ABB RobotStudio station: Topsy_Turvey_Pack_N_Go_RW_5.16.rspag

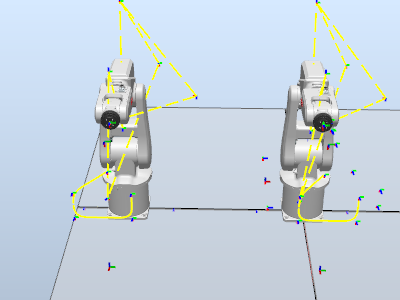
--- station ---
Station Turvey_Solution_2 (saved by RobotStudio 24.2.10789.0)
Controller 120-502354_Topsy, task T_ROB1: task frame (RAPID world) sits at (0, -769, 0) mm in the station
Controller 120-501650_Turvey
  mechanical unit ROB_1: IRB120_Turvey, 6 joints, base frame (0, 0, 0) mm
Controller 120-502354_Topsy
  mechanical unit ROB_1: IRB120_Topsy, 6 joints, base frame (0, 0, 0) mm
Layout (positions relative to the parent item):
  - IRB120_Turvey [mechanism, from %ABB.RobotStudio.Models.IRB120%\IRB120_3_58_G_01.rslib] at (0, 0, 0) mm; joint values [0, 0, 0, 0, 0, 0] (rad or m)
  - IRB120_Topsy [mechanism, from %ABB.RobotStudio.Models.IRB120%\IRB120_3_58_G_01.rslib] at (0, -769, 0) mm; joint values [0, 0, 0, 0, 0, 0] (rad or m)
Targets, tools, work objects and paths stored in the station and not in the controller backup, written as RAPID:
! task T_ROB1
MODULE MainModule
  CONST robtarget pos1:=[[366.18,1.37,632.09],[0.674845,-0.0204665,0.737511,-0.015567],[0,0,-1,0],[9E+09,9E+09,9E+09,9E+09,9E+09,9E+09]];
  CONST jointtarget JtCalpos:=[[0,0,0,0,0,0],[9E+09,9E+09,9E+09,9E+09,0,9E+09]];
  CONST jointtarget JtHome:=[[0,0,0,90,0,0],[9E+09,9E+09,9E+09,9E+09,0,9E+09]];
  PROC R_Home()
    WaitTime 5;
    WaitTime 5;
    MoveAbsJ jHomePos,v500,fine,tool0;
  ENDPROC
  PROC R_Storage()
    WaitTime 5;
    WaitTime 5;
    MoveAbsJ jStorage,v500,fine,tool0;
  ENDPROC
ENDMODULE

! task T_ROB1
MODULE MainModule
  PROC R_Home()
    WaitTime 5;
    WaitTime 5;
    MoveAbsJ jHomePos,v500,fine,tool0;
  ENDPROC
  PROC R_Storage()
    WaitTime 5;
    WaitTime 5;
    MoveAbsJ jStorage,v500,fine,tool0;
  ENDPROC
ENDMODULE


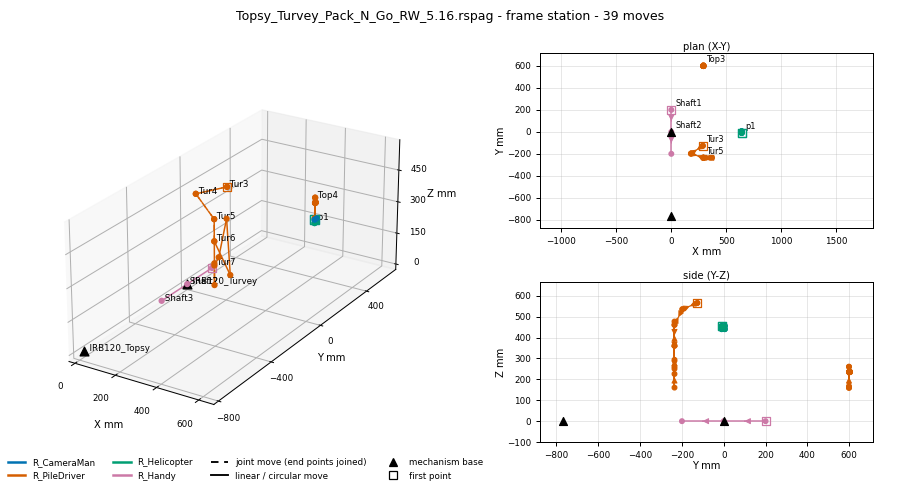
[picture p0: tool path of Topsy_Turvey_Pack_N_Go_RW_5.16.rspag in frame station, 39 of 203 moves have a stored position in this frame; points joined in program order, loops and branches not executed]
--- Backups/120-501650_Turvey/RAPID/TASK1/PROGMOD/MainModule.mod ---
MODULE MainModule
    !    !*****************************************************
    !    !Module Name:   MainModule
    !    !Version:       1.22
    !    !Description:   Main Module
    !    !Date:          2024-08-01
    !    !Author:        @ManicZanic
    !    !*****************************************************
    !    !Change Log:
    !    !2024-08-01:    @ManicZanic - Orignal core structure developed
    !    !2024-08-21:    @ManicZanic - Moved non TOH routines to Main module.
    !    !                           - Added Menu options to all routines.
    !    !                           - Added NCameraLoop to disconnect variables from other modules
    !    !                           - Cleaned up text a bit
    !    !                           - Formatted text
    !    !                           - Added Yoga Pose positions
    !    !                           - Added blank JustDance program
    !    !2024-08-22:    @ManicZanic - Removed unused code
    !    !                           - Removed task specific ToolData
    !    !2024-08-22:    @ManicZanic - Programmed DancingQueen routine.
    !    !                           - Programmed YogaPose routine
    !    !                           - Edited menu names
    !    !2024-08-26:    @ManicZanic - Modified motion alert notification interface.
    !    !                           - Created universal speed selection progam
    !    !                           - Modified Yoga Poses
    !    !2024-08-29:    @ManicZanic - Updated UI to add option for no motion alarm and to edit menus
    !    !*****************************************************

    PERS bool bMenu:=TRUE;
    PERS bool bTopsy:=FALSE;
    PERS bool bTurvey:=TRUE;
    PERS bool CondomMode:=FALSE;
    PERS bool RawDogMode:=TRUE;

    !CURRENT VELOCITY
    VAR speeddata VSpeed:=V300;

    VAR num ERR_TP_DOBREAK;
    !VAR num CurrentIndex:=nMenuOption;
    VAR num nMenuOption;

    VAR btnres answer;

    CONST string LoopMessage{5}:=[" "," ","Enter How Many Times To Loop Dance Program"," ","0=INFINITE"];
    CONST string CautionMessage{5}:=[" "," "," ","Press RUN to continue","Press CANCEL to return to previous menu"];
    CONST string RunCancel{2}:=["RUN","CANCEL"];
    CONST string MenuButtons{5}:=["SET SPEED","MENU","","RUN","CANCEL"];

    PERS tooldata tMain:=[TRUE,[[0.000145392,0,140.499655058],[1,0,-0.000000126,0]],[1,[0,0,75],[1,0,0,0],0,0,0]];

    CONST jointtarget jHomePos:=[[0,0,0,0,0,0],[9E+09,9E+09,9E+09,9E+09,9E+09,9E+09]];
    CONST jointtarget jStorage:=[[0,0,-90,0,0,0],[9E+09,9E+09,9E+09,9E+09,9E+09,9E+09]];
    CONST jointtarget jDongStoragePos:=[[90,0,0,0,90,0],[9E+09,9E+09,9E+09,9E+09,9E+09,9E+09]];


    PROC Main()
        SafeModeMenu;
    ENDPROC




    PROC SafeModeMenu()
        VAR num nMenuOption;
        VAR btnres btnresMainMenu;
        CONST Listitem ListOptions{6}:=[
        ["1","WANNA SEE SOMETHING COOL!!!"],
        ["2","Select a mode and press OK"],
        ["3"," "],
        ["4","Kid Mode"],
        ["5","Big Boy Dont Need No Warning Mode"],
        ["6",""]];

        bMenu:=True;
        WHILE bMenu DO
            nMenuOption:=UIListView(\Result:=btnresMainMenu\Header:="Please select an option and press OK",ListOptions\Buttons:=btnOkCancel\Icon:=iconInfo);
            IF btnresMainMenu=resCancel Main;
            TEST nMenuOption
            CASE 4:
                CondomMode:=TRUE;
                Main_Menu;
            CASE 5:
                CondomMode:=FALSE;
                Main_Menu;

            ENDTEST
        ENDWHILE
        bMenu:=TRUE;
    ENDPROC


    PROC Main_Menu()
        VAR num nMenuOption;
        VAR btnres btnresMainMenu;
        VAR num Temp1:=0;
        CONST Listitem ListOptions{18}:=[
            ["1","Set Speed"],
            ["2","Home Position"],
            ["3","Dong Storage Position"],
            ["4","Storage Position"],
            ["5","Camera Man"],
            ["6","Yoga Pose"],
            ["7","Just Dance"],
            ["8","Tower of Hanoi"],
            ["9","Helicopter Helicopter"],
            ["10","Pile Driver"],
            ["11"," "],
            ["12","***DONT LOOK IM NOT CODED YET!!!***"],
            ["13 to be declared in slot 11","Docking"],
            ["14",""],
            ["15"," "],
            ["16"," "],
            ["17"," "],
            ["18"," "]];

        bMenu:=True;
        WHILE bMenu DO
            nMenuOption:=UIListView(\Result:=btnresMainMenu\Header:="Please select an option and press OK",ListOptions\Btnarray:=MenuButtons\Icon:=iconInfo);
            IF btnresMainMenu=1 R_Set_SPEEEEEED;
            IF btnresMainMenu=2 RawdogMode:=FALSE;
            IF btnresMainMenu=4 RawdogMode:=TRUE;
            IF btnresMainMenu=5 Main_Menu;


            TEST nMenuOption
            CASE 1:
                R_Set_SPEEEEEED;
                Main_Menu;
            CASE 2:
                IF CondomMode=TRUE THEN
                    answer:=UIMessageBox(\Header:="CAUTION: ROBOT MAY MOVE"\MsgArray:=CautionMessage\BtnArray:=RunCancel\Icon:=IconWarning);
                    IF answer=1 THEN
                        MoveAbsJ jHomePos,v150,fine,tool0;
                    ELSEIF answer=2 THEN
                        Main_Menu;
                    ENDIF
                ELSE
                    MoveAbsJ jHomePos,v150,fine,tool0;
                ENDIF
            CASE 3:
                IF CondomMode=TRUE THEN
                    answer:=UIMessageBox(\Header:="CAUTION: ROBOT MAY MOVE"\MsgArray:=CautionMessage\BtnArray:=RunCancel\Icon:=IconWarning);
                    IF answer=1 THEN
                        MoveAbsJ jDongStoragePos,v150,fine,tool0;
                    ELSEIF answer=2 THEN
                        Main_Menu;
                    ENDIF
                ELSE
                    MoveAbsJ jDongStoragePos,v150,fine,tool0;
                    Main_Menu;
                ENDIF
            CASE 4:
                IF CondomMode=TRUE THEN
                    answer:=UIMessageBox(\Header:="CAUTION: ROBOT MAY MOVE"\MsgArray:=CautionMessage\BtnArray:=RunCancel\Icon:=IconWarning);
                    IF answer=1 THEN
                        MoveAbsJ jStorage,v150,fine,tool0;
                    ELSEIF answer=2 THEN
                        Main_Menu;
                    ENDIF
                ELSE
                    MoveAbsJ jStorage,v150,fine,tool0;
                ENDIF
                Main_Menu;

            CASE 5:
                IF RawDogMode=FALSE THEN
                    R_CameraMan_Menu;
                ELSE
                    NCameraLoop:=2;
                    R_CameraMan;
                ENDIF
            CASE 6:
                IF RawDogMode=FALSE THEN
                    R_YogaPose;
                ELSE
                    MoveAbsJ jCobra,v150,fine,tool0;
                    WaitTime 5;
                    MoveAbsJ jDoggyStyle,v150,fine,tool0;
                    WaitTime 5;
                    MoveAbsJ jCamel,v150,fine,tool0;
                    WaitTime 5;
                    MoveAbsJ jChair,v150,fine,tool0;
                    WaitTime 5;
                    MoveAbsJ jStarGazer,v150,fine,tool0;
                    TPErase;
                    TPWrite "HEY LOOK A ROCKET SHIP";
                    WaitTime 2;
                    TPWrite "*      *      *";
                    TPWrite "*    *       *    *";
                    TPWrite "   8=====D~~...___";
                    TPWrite "*      *      *";
                    TPWrite "*    *       *    *";
                    WaitTime 5;
                    TPErase;

                ENDIF
            CASE 7:
                IF RawDogMode=FALSE THEN
                    R_DancingQueen_Menu;
                ELSE
                    R_DancingQueen;
                ENDIF
            CASE 8:
                IF RawDogMode=FALSE THEN
                    %"R_Tower_Of_Hanoi_Menu"%;
                ELSE
                    %"R_Tower_Of_Hanoi_SolSel"%;
                ENDIF
            CASE 9:
                IF RawDogMode=FALSE THEN
                    R_Helicopter_Menu;
                ELSE
                    nHelicopter:=2;
                    R_Helicopter;
                ENDIF
            CASE 10:
                IF RawDogMode=FALSE THEN
                    R_PileDriver_Menu;
                ELSE
                    R_PileDriver;
                ENDIF
            CASE 11:
                IF RawDogMode=FALSE THEN
                    R_Docking_Menu;
                ELSE
                    R_Docking;
                ENDIF

            CASE 12:
                TPErase;
                TPWrite "***PERVERT***";
                WaitTime 2;
                TPerase;
                RETURN ;
                bMenu:=False;
            ENDTEST
        ENDWHILE
        bMenu:=TRUE;
    ENDPROC

    PROC R_Set_SPEEEEEED()
        VAR num nMenuOption;
        VAR btnres btnresMainMenu;
        VAR num change_speed:=60;

        CONST Listitem ListOptions{7}:=[
        ["","Super Slow"],
        ["","Slow"],
        ["","Normal"],
        ["","Fast"],
        ["","Super Fast"],
        ["","Helicopter"],
        ["","JUST DONT!!!"]];

        bMenu:=True;
        WHILE bMenu DO
            nMenuOption:=UIListView(\Result:=btnresMainMenu\Header:="Select Desired Speed",ListOptions\Buttons:=btnOKCancel\Icon:=iconInfo);
            IF btnresMainMenu=resCancel RETURN;
            TEST nMenuOption
            CASE 1:
                VSpeed:=V150;
                RETURN ;
            CASE 2:
                VSpeed:=V300;
                RETURN ;
            CASE 3:
                VSpeed:=V500;
                RETURN ;
            CASE 4:
                VSpeed:=V1000;
                RETURN ;
            CASE 5:
                VSpeed:=V2500;
                RETURN ;
            CASE 6:
                VSpeed:=V300;
                SpeedRefresh change_speed;
                RETURN ;
            CASE 7:
                VSpeed:=V10;
                RETURN ;
                !SpeedRefresh change_speed;
                bMenu:=False;
            ENDTEST
        ENDWHILE
        bMenu:=True;
    ENDPROC
ENDMODULE

--- Backups/120-501650_Turvey/RAPID/TASK1/PROGMOD/M_CameraMan.mod ---
MODULE M_CameraMan
    !    !*****************************************************
    !    !Module Name:   M_TEMPLATE
    !    !Version:       1.22
    !    !Description:   CameraMan
    !    !Date:          2024-08-30
    !    !Author:        @ManicZanic
    !    !
    !    !*****************************************************
    !    !Change Log:
    !    !2024-08-31:    @ManicZanic - Orignal core pulled from MainModule
    !    !*****************************************************

    !CAMERAMAN LOOP SWITCH
    PERS num NCameraLoop:=1;

    PROC R_CameraMan_Menu()
        VAR num nMenuOption;
        VAR btnres btnresMainMenu;
        CONST Listitem ListOptions{7}:=[
        ["1","Select an option and press OK to run program"],
            ["2","Press CANCEL to return to Main Menu"],
            ["3"," "],
            ["4"," "],
            ["5","Set Speed"],
            ["6"," "],
            ["7","RUN PROGRAM"]];
        !       Menu Start
        bMenu:=True;
        WHILE bMenu DO
            nMenuOption:=UIListView(\Result:=btnresMainMenu\Header:="RUN CAMERAMAN PROGRAM",ListOptions\Buttons:=btnOKCancel\Icon:=iconWarning);
            IF btnresMainMenu=resCancel Main_Menu;
            TEST nMenuOption
            CASE 1:
                TPErase;
                TPwrite "Wrong hole...WRONG HOLE!!!!!";
                waittime 5;
                TPErase;
            CASE 2:
                TPErase;
                TPwrite "Wrong hole...WRONG HOLE!!!!!";
                waittime 5;
                TPErase;
                Main_Menu;
            CASE 3:
            CASE 4:
            CASE 5:
                R_Set_SPEEEEEED;
                R_CameraMan_Menu;
            CASE 6:
            CASE 7:
                IF CondomMode=TRUE THEN
                    answer:=UIMessageBox(\Header:="CAUTION: ROBOT MAY MOVE"\MsgArray:=CautionMessage\BtnArray:=RunCancel\Icon:=IconWarning);
                    IF answer=1 THEN
                        NCameraLoop:=2;
                        R_CameraMan;
                        Main_Menu;
                    ELSEIF answer=2 THEN
                        Main_Menu;
                    ENDIF
                ELSE
                    NCameraLoop:=2;
                    R_CameraMan;
                    Main_Menu;
                ENDIF
                Main_Menu;
                bMenu:=False;
            ENDTEST
        ENDWHILE
    ENDPROC

    PROC R_CameraMan()
        CONST jointtarget jCameraMan:=[[0,26.8166,-4.77057,0,-22.0461,0],[9E+09,9E+09,9E+09,9E+09,9E+09,9E+09]];
        CONST robtarget p1:=[[640.50,-10,455.00],[0.707107,3.47691E-8,0.707107,-1.5478E-9],[-1,-1,0,1],[9E+9,9E+9,9E+9,9E+9,9E+9,9E+9]];
        CONST robtarget p2:=[[640.50,-10,440.00],[0.707107,7.61395E-9,0.707107,7.08051E-9],[-1,-1,0,1],[9E+9,9E+9,9E+9,9E+9,9E+9,9E+9]];
        CONST robtarget p3:=[[640.50,5,440.00],[0.707107,-7.61395E-9,0.707107,-7.08051E-9],[0,0,-1,1],[9E+9,9E+9,9E+9,9E+9,9E+9,9E+9]];
        CONST robtarget p4:=[[640.50,5,455.00],[0.707107,-3.47691E-8,0.707107,1.5478E-9],[0,0,-1,1],[9E+9,9E+9,9E+9,9E+9,9E+9,9E+9]];

        IF NCameraLoop=2 THEN
            MoveAbsJ jCameraMan,v500,fine,tMain;
            NCameraLoop:=1;
            setdo SOManButt_on4, 1;
        ENDIF
!        WHILE TRUE DO
        WHILE DOutput(SOManButt_on4)=1 DO
        MoveL p1,vSpeed,z50,tMain;
        MoveL p2,vSpeed,z50,tMain;
        MoveL p3,vSpeed,z50,tMain;
        MoveL p4,vSpeed,z50,tMain;
        ENDWHILE
        RETURN;
    ENDPROC
ENDMODULE

--- Backups/120-501650_Turvey/RAPID/TASK1/PROGMOD/M_DancingQueen.mod ---
MODULE M_DancingQueen
    !    !*****************************************************
    !    !Module Name:   M_TEMPLATE
    !    !Version:       1.22
    !    !Description:   DancingQueen
    !    !Date:          2024-08-30
    !    !Author:        @ManicZanic
    !    !
    !    !*****************************************************
    !    !Change Log:
    !    !2024-08-30:    @ManicZanic - Core structure pulled from MainModule
    !    !*****************************************************

    VAR num NDanceLoop:=1;
    VAR num NCurrentDanceLoop:=0;

    PROC R_DancingQueen_Menu()
        VAR num nMenuOption;
        VAR btnres btnresMainMenu;
        CONST Listitem ListOptions{7}:=[["1","Select an option and press OK to run program"],["2","Press CANCEL to return to Main Menu"],[""," "],[""," "],["","SET SPEED"],["","SET LOOP"],["","RUN PROGRAM"]];
        !       Menu Start
        bMenu:=True;
        WHILE bMenu DO
            nMenuOption:=UIListView(\Result:=btnresMainMenu\Header:="RUN DANCING QUEEN",ListOptions\Buttons:=btnOKCancel\Icon:=iconWarning);
            IF btnresMainMenu=resCancel Main_Menu;
            TEST nMenuOption
            CASE 1:
                TPErase;
                TPwrite "Wrong hole...WRONG HOLE!!!!!";
                waittime 5;
                TPErase;
            CASE 2:
                TPErase;
                TPwrite "Wrong hole...WRONG HOLE!!!!!";
                waittime 5;
                TPErase;
                RETURN ;
            CASE 3:
            CASE 4:
            CASE 5:
                R_Set_SPEEEEEED;
                R_DancingQueen_Menu;
            CASE 6:
                NDanceLoop:=UINumEntry(\Header:="Set Repeat Counter"\MsgArray:=LoopMessage\Icon:=iconInfo\InitValue:=NDanceLoop\MinValue:=0\MaxValue:=1000);
                R_DancingQueen_Menu;
            CASE 7:
                answer:=UIMessageBox(\Header:="CAUTION: ROBOT MAY MOVE"\MsgArray:=CautionMessage\BtnArray:=RunCancel\Icon:=IconWarning);
                IF answer=1 THEN
                    NCurrentDanceLoop:=0;
                    R_DancingQueen;
                ELSEIF answer=2 THEN
                    RETURN ;
                ENDIF
                Main_Menu;
                bMenu:=False;
            ENDTEST
        ENDWHILE
    ENDPROC

    PROC R_DancingQueen()
        CONST jointtarget j1:=[[0,0,-90,0,0,0],[9E+09,9E+09,9E+09,9E+09,9E+09,9E+09]];
        CONST jointtarget j2:=[[45,-34.7368,0,30,-45,0],[9E+09,9E+09,9E+09,9E+09,9E+09,9E+09]];
        CONST jointtarget j3:=[[-45,-35,0,-30,-45,0],[9E+09,9E+09,9E+09,9E+09,9E+09,9E+09]];
        CONST jointtarget j4:=[[45,-33.512,43.8106,8.56333E-05,-10.2984,-8.82129E-05],[9E+09,9E+09,9E+09,9E+09,9E+09,9E+09]];
        CONST jointtarget j5:=[[45,29.6234,-17.5512,3.19074E-05,-12.0721,-3.12018E-05],[9E+09,9E+09,9E+09,9E+09,9E+09,9E+09]];
        CONST jointtarget j6:=[[-45,-33.4907,43.6889,-7.08038E-05,-10.2336,-0.320042],[9E+09,9E+09,9E+09,9E+09,9E+09,9E+09]];
        CONST jointtarget j7:=[[-45,29.6402,-17.6857,-5.55671E-05,-11.99,-0.320058],[9E+09,9E+09,9E+09,9E+09,9E+09,9E+09]];
        CONST jointtarget j8:=[[45,19.6394,40.4538,2.45022E-06,-60.0932,-1.22166E-06],[9E+09,9E+09,9E+09,9E+09,9E+09,9E+09]];
        CONST jointtarget j9:=[[-45,19.6394,40.4538,2.45022E-06,-60.0932,-1.22166E-06],[9E+09,9E+09,9E+09,9E+09,9E+09,9E+09]];
        CONST jointtarget j10:=[[45,0,0,0,0,0],[9E+09,9E+09,9E+09,9E+09,9E+09,9E+09]];
        CONST jointtarget j11:=[[45,0,0,0,0,0],[9E+09,9E+09,9E+09,9E+09,9E+09,9E+09]];
        CONST jointtarget j12:=[[45,0,0,0,0,0],[9E+09,9E+09,9E+09,9E+09,9E+09,9E+09]];
        CONST jointtarget j13:=[[45,0,0,0,0,0],[9E+09,9E+09,9E+09,9E+09,9E+09,9E+09]];
        CONST jointtarget j14:=[[45,0,0,0,0,0],[9E+09,9E+09,9E+09,9E+09,9E+09,9E+09]];
        CONST jointtarget j15:=[[45,0,0,0,0,0],[9E+09,9E+09,9E+09,9E+09,9E+09,9E+09]];
        CONST jointtarget j16:=[[45,0,0,0,0,0],[9E+09,9E+09,9E+09,9E+09,9E+09,9E+09]];
        CONST jointtarget j17:=[[45,0,0,0,0,0],[9E+09,9E+09,9E+09,9E+09,9E+09,9E+09]];
        CONST jointtarget j18:=[[45,0,0,0,0,0],[9E+09,9E+09,9E+09,9E+09,9E+09,9E+09]];
        CONST jointtarget j19:=[[45,0,0,0,0,0],[9E+09,9E+09,9E+09,9E+09,9E+09,9E+09]];
        CONST jointtarget j20:=[[45,0,0,0,0,0],[9E+09,9E+09,9E+09,9E+09,9E+09,9E+09]];


        MoveAbsJ j1,VSpeed,fine,tool0;
        MoveAbsJ j2,VSpeed,fine,tool0;
        MoveAbsJ j1,VSpeed,fine,tool0;
        MoveAbsJ j2,VSpeed,fine,tool0;
        MoveAbsJ j1,VSpeed,fine,tool0;
        MoveAbsJ j3,VSpeed,fine,tool0;
        MoveAbsJ j1,VSpeed,fine,tool0;
        MoveAbsJ j3,VSpeed,fine,tool0;
        MoveAbsJ j1,VSpeed,fine,tool0;
        MoveAbsJ j4,VSpeed,fine,tool0;
        MoveAbsJ j1,VSpeed,fine,tool0;
        MoveAbsJ j4,VSpeed,fine,tool0;
        MoveAbsJ j1,VSpeed,fine,tool0;
        MoveAbsJ j5,VSpeed,fine,tool0;
        MoveAbsJ j1,VSpeed,fine,tool0;
        MoveAbsJ j5,VSpeed,fine,tool0;
        MoveAbsJ j1,VSpeed,fine,tool0;
        MoveAbsJ j6,VSpeed,fine,tool0;
        MoveAbsJ j1,VSpeed,fine,tool0;
        MoveAbsJ j6,VSpeed,fine,tool0;
        MoveAbsJ j1,VSpeed,fine,tool0;
        MoveAbsJ j7,VSpeed,fine,tool0;
        MoveAbsJ j1,VSpeed,fine,tool0;
        MoveAbsJ j7,VSpeed,fine,tool0;
        MoveAbsJ j1,VSpeed,fine,tool0;
        MoveAbsJ j8,VSpeed,fine,tool0;
        MoveAbsJ j1,VSpeed,fine,tool0;
        MoveAbsJ j8,VSpeed,fine,tool0;
        MoveAbsJ j1,VSpeed,fine,tool0;
        MoveAbsJ j9,VSpeed,fine,tool0;
        MoveAbsJ j1,VSpeed,fine,tool0;
        MoveAbsJ j9,VSpeed,fine,tool0;
        MoveAbsJ j8,VSpeed,fine,tool0;
        MoveAbsJ j9,VSpeed,fine,tool0;
        MoveAbsJ j8,VSpeed,fine,tool0;
        MoveAbsJ j9,VSpeed,fine,tool0;
        MoveAbsJ j6,VSpeed,fine,tool0;
        MoveAbsJ j7,VSpeed,fine,tool0;
        MoveAbsJ j6,VSpeed,fine,tool0;
        MoveAbsJ j7,VSpeed,fine,tool0;
        MoveAbsJ j6,VSpeed,fine,tool0;
        MoveAbsJ j4,VSpeed,fine,tool0;
        MoveAbsJ j5,VSpeed,fine,tool0;
        MoveAbsJ j4,VSpeed,fine,tool0;
        MoveAbsJ j5,VSpeed,fine,tool0;
        MoveAbsJ j4,VSpeed,fine,tool0;
        MoveAbsJ j2,VSpeed,fine,tool0;
        MoveAbsJ j3,VSpeed,fine,tool0;
        MoveAbsJ j2,VSpeed,fine,tool0;
        MoveAbsJ j3,VSpeed,fine,tool0;
        MoveAbsJ j1,VSpeed,fine,tool0;
        Incr NCurrentDanceLoop;
        IF NDanceLoop=0 OR NDanceLoop>NCurrentDanceLoop THEN
            R_DancingQueen;
        ENDIF
        MoveAbsJ jHomePos\NoEOffs,VSpeed,fine,tool0;
        !Place Code Here
    ENDPROC

ENDMODULE

--- Backups/120-501650_Turvey/RAPID/TASK1/PROGMOD/M_DirtyDeeds.mod ---
MODULE M_DirtyDeeds
    !    !*****************************************************
    !    !Module Name:   M_TEMPLATE
    !    !Version:       1.22
    !    !Description:   DirtyDeeds
    !    !Date:          2024-08-30
    !    !Author:        @ManicZanic
    !    !
    !    !*****************************************************
    !    !Change Log:
    !    !2024-08-30:    @ManicZanic - Orignal core structure developed
    !    !2024-09-01:    @ManicZanic - modifed piledriver program
    !    !*****************************************************


    VAR num NThrustLoop:=50;
    VAR num NCurrentThrustLoop:=0;
    VAR num NThrustTemp1:=0;
    VAR num NThrustTemp2:=0;
    VAR num NThrustTemp3:=0;
    VAR num NThrustTemp4:=0;
    VAR num NThrustTemp5:=0;
    VAR num NThrustTemp6:=0;
    VAR num NThrustTemp7:=0;
    CONST string ThrustMessage{6}:=[" ","Enter How Many Strokes to Achieve 'Completion'"," ","NOTE: Actual stroke limits are calculated an may differ from specified number"," ","0=Cialis Mode"];
    CONST string DTFTurMessage{10}:=["Are you ready Baby"," "," ","NOTE: Press YES on both controllers at the same time"," "," ","By pressing Yes this robot concents to the"," following actions of its own 'free will'.","At any time this robot can relinquish its concent","by exiting the while command"];
    CONST string DTFTopMessage{10}:=["Is that what I think it is?"," ","NOTE: Press YES on both controllers at the same time"," "," ","By pressing Yes this robot concents to the"," "," following actions of its own 'free will'.","At any time this robot can relinquish its concent","by exiting the while command"];
    CONST string DTFCompletionMessage{5}:=["Was it good for you"," ","NOTE: Press either option on both controllers at the same time","To send the robots back home.","This message can be removed once IO is established"];
    CONST string DTFTurButtons{2}:=["YES Daddy","I Have A Headache"];
    CONST string DTFTopButtons{2}:=["YES ","I Have A Headache"];
    CONST string DTFCompletionButtons{2}:=["THAT WAS AMAZING","Maybe next time"];
    VAR num Thrust_Speed:=100;

    PERS tooldata tDong:=[TRUE,[[0.000145392,0,140.499655058],[1,0,-0.000000126,0]],[1,[0,0,75],[1,0,0,0],0,0,0]];


    PROC R_PileDriver_Menu()
        VAR num nMenuOption;
        VAR btnres btnresMainMenu;
        CONST Listitem ListOptions{7}:=[
        ["1","Select an option and press OK to run program"],
        ["2","Press CANCEL to return to Main Menu"],
        [""," "],
        [""," "],
        ["","SET SPEED"],
        ["","SET THRUST COUNT"],
        ["","RUN PROGRAM"]];
        !       Menu Start
        bMenu:=True;
        WHILE bMenu DO
            nMenuOption:=UIListView(\Result:=btnresMainMenu\Header:="PILE DRIVER MENU",ListOptions\Buttons:=btnOKCancel\Icon:=iconWarning);
            IF btnresMainMenu=resCancel Main_Menu;
            TEST nMenuOption
            CASE 1:
                TPErase;
                TPwrite "Wrong hole...WRONG HOLE!!!!!";
                waittime 5;
                TPErase;
            CASE 2:
                TPErase;
                TPwrite "Wrong hole...WRONG HOLE!!!!!";
                waittime 5;
                TPErase;
                RETURN ;
            CASE 3:
            CASE 4:
            CASE 5:
                R_Set_SPEEEEEED;
                R_PileDriver_Menu;
            CASE 6:
                NThrustLoop:=UINumEntry(\Header:="Set Thrust Counter"\MsgArray:=ThrustMessage\Icon:=iconInfo\InitValue:=NThrustLoop\MinValue:=0\MaxValue:=1000);
                R_PileDriver_Menu;
            CASE 7:
                IF CondomMode=TRUE THEN
                answer:=UIMessageBox(\Header:="CAUTION: ROBOT MAY MOVE"\MsgArray:=CautionMessage\BtnArray:=RunCancel\Icon:=IconWarning);
                IF answer=1 THEN
                    NCurrentThrustLoop:=0;
                    R_PileDriver;
                ELSEIF answer=2 THEN
                    R_PileDriver_Menu;
                ENDIF
                ELSE
                    NCurrentThrustLoop:=0;
                    R_PileDriver;
                ENDIF

                bMenu:=False;
                Main_Menu;
            ENDTEST
        ENDWHILE
    ENDPROC

    PROC R_PileDriver()

        CONST jointtarget JLimpDick:=[[45,-34.7368,0,30,-45,0],[9E+09,9E+09,9E+09,9E+09,9E+09,9E+09]];
        CONST jointtarget jTur1:=[[0,0,0,0,0,0],[9E+09,9E+09,9E+09,9E+09,9E+09,9E+09]];
        CONST jointtarget jTur2:=[[-2.8048,-2.01481,-20.6326,-5.72958E-05,78.3158,87.1952],[9E+09,9E+09,9E+09,9E+09,9E+09,9E+09]];
        CONST robtarget Tur3:=[[286.92,-126.72,565.24],[0.218656,0.675608,0.675609,0.198231],[-1,0,0,0],[9E+09,9E+09,9E+09,9E+09,9E+09,9E+09]];
        CONST robtarget Tur4:=[[178.47,-197.92,535.20],[0.00090867,0.707358,0.706855,0.00012926],[-1,0,0,0],[9E+09,9E+09,9E+09,9E+09,9E+09,9E+09]];
        CONST robtarget Tur5:=[[292.64,-235.68,460.54],[0.000909492,0.707358,0.706855,0.000129512],[-1,0,0,0],[9E+09,9E+09,9E+09,9E+09,9E+09,9E+09]];
        CONST robtarget Tur6:=[[292.64,-235.68,360.54],[0.000909428,0.707358,0.706855,0.000129512],[-1,0,0,0],[9E+09,9E+09,9E+09,9E+09,9E+09,9E+09]];
        CONST robtarget Tur7:=[[292.64,-235.68,250.54],[0.0317414,0.706679,0.706142,0.0309839],[-1,0,0,0],[9E+09,9E+09,9E+09,9E+09,9E+09,9E+09]];
        CONST robtarget Tur8:=[[314.24,-235.68,293.36],[0.0807965,0.70281,0.702223,0.0800788],[-1,0,0,0],[9E+09,9E+09,9E+09,9E+09,9E+09,9E+09]];
        CONST robtarget Tur9:=[[353.21,-235.68,476.43],[0.155776,0.690138,0.689478,0.155125],[-1,0,0,0],[9E+09,9E+09,9E+09,9E+09,9E+09,9E+09]];
        CONST robtarget Tur10:=[[370.66,-235.68,225.83],[0.192165,0.680928,0.680234,0.19155],[-1,0,0,0],[9E+09,9E+09,9E+09,9E+09,9E+09,9E+09]];

        CONST jointtarget jTop1:=[[0,0,0,0,0,0],[9E+09,9E+09,9E+09,9E+09,9E+09,9E+09]];
        CONST jointtarget jTop2:=[[37.4546,30.9643,39.4089,-54.5501,-78.2187,105.821],[9E+09,9E+09,9E+09,9E+09,9E+09,9E+09]];
        CONST robtarget Top3:=[[291.87,598.76,160.24],[0.00175179,0.00248362,-0.707669,-0.706538],[0,-1,1,1],[9E+09,9E+09,9E+09,9E+09,9E+09,9E+09]];
        CONST robtarget Top4:=[[291.87,598.76,260.24],[0.00175187,0.00248369,-0.707669,-0.706538],[0,-1,1,1],[9E+09,9E+09,9E+09,9E+09,9E+09,9E+09]];
        !        CONST robtarget Top5:=[[293.04,498.76,360.53],[0.498863,-0.49923,0.500893,0.501011],[0,1,-2,0],[9E+09,9E+09,9E+09,9E+09,9E+09,9E+09]];
        !        CONST robtarget Top6:=[[293.04,498.76,360.53],[0.498863,-0.49923,0.500893,0.501011],[0,1,-2,0],[9E+09,9E+09,9E+09,9E+09,9E+09,9E+09]];

        IF NThrustLoop>10 THEN
            NThrustTemp1:=Round(NThrustLoop/7);
            NThrustTemp2:=nthrustTemp1+NThrustTemp1;
            NThrustTemp3:=nthrustTemp2+NThrustTemp1;
            NThrustTemp4:=nthrustTemp3+NThrustTemp1;
            NThrustTemp5:=nthrustTemp4+NThrustTemp1;
            NThrustTemp6:=nthrustTemp5+NThrustTemp1;
            NThrustTemp7:=nthrustTemp6+NThrustTemp1;
            Nthrustloop:=Nthrusttemp7;
        ELSE
            NThrustTemp1:=2;
            NThrustTemp2:=3;
            NThrustTemp3:=4;
            NThrustTemp4:=5;
            NThrustTemp5:=6;
            NThrustTemp6:=8;
            NThrustTemp7:=10;
        ENDIF
        IF bTurvey=TRUE AND bTopsy=FALSE THEN
            MoveAbsJ jTur1,VSpeed,fine,tDong;
            MoveAbsJ jTur2,VSpeed,fine,tDong;
            MoveJ Tur3,vSpeed,z50,tDong;
            MoveJ Tur4,vSpeed,z50,tDong;
            MoveJ Tur5,vSpeed,z50,tDong;
            MoveL Tur6,vSpeed,fine,tDong;
            answer:=UIMessageBox(\Header:="Do I Make You Horney Baby? YEAAA!!!"\MsgArray:=DTFTurMessage\BtnArray:=DTFTurButtons\Icon:=IconWarning);
            IF answer=1 THEN
                NCurrentThrustLoop:=0;
                WHILE NThrustLoop>NCurrentThrustLoop DO
                    IF NcurrentthrustLoop=1 THEN
                        TPErase;
                        TPwrite "You like that don't you.";
                        Thrust_Speed:=30;
                        SpeedRefresh Thrust_Speed;
                    ENDIF
                    IF NcurrentthrustLoop=NThrustTemp3 THEN
                        Thrust_Speed:=40;
                        SpeedRefresh Thrust_Speed;
                    ENDIF
                    IF NcurrentthrustLoop=NThrustTemp4 THEN
                        Thrust_Speed:=50;
                        SpeedRefresh Thrust_Speed;
                    ENDIF
                    IF NcurrentthrustLoop=NThrustTemp5 THEN
                        Thrust_Speed:=75;
                        SpeedRefresh Thrust_Speed;
                    ENDIF
                    IF NcurrentthrustLoop=NThrustTemp6 THEN
                        Thrust_Speed:=100;
                        SpeedRefresh Thrust_Speed;
                    ENDIF
                    MoveL offs(Tur6,0,0,-200),VSpeed,fine,tDong;
                    MoveL offs(Tur6,0,0,-100),VSpeed,fine,tDong;
                    Incr NCurrentThrustLoop;
                    IF NcurrentthrustLoop=NThrustTemp7 THEN
                        TPwrite "BEEP BOP BOOP";
                        WaitTime 1;
                        TPwrite "---I HAVE ARIVED---";
                        WaitTime 1;
                        Thrust_Speed:=50;
                        SpeedRefresh Thrust_Speed;
                        MoveL Tur7,vSpeed,fine,tDong;
                        MoveL Tur8,vSpeed,z50,tDong;
                        MoveL Tur9,vSpeed,z50,tDong;
                        MoveL Tur10,vSpeed,fine,tDong;
                        TPwrite "Now go get yourself cleaned up.";
                    ENDIF
                ENDWHILE
                answer:=UIMessageBox(\Header:="Was it good for you"\MsgArray:=DTFCompletionMessage\BtnArray:=DTFCompletionButtons\Icon:=IconWarning);
                IF answer=1 THEN
                ENDIF
                MoveL Tur6,vSpeed,z50,tDong;
                MoveJ Tur5,vSpeed,z50,tDong;
                MoveJ Tur4,vSpeed,z50,tDong;
                MoveJ Tur3,vSpeed,z50,tDong;
                MoveAbsJ jTur2,VSpeed,fine,tDong;
                MoveAbsJ jTur1,VSpeed,fine,tDong;
                !                ENDIF
            ELSEIF answer=2 THEN
                MoveAbsJ jLimpDick,VSpeed,fine,tool0;
            ENDIF
            MoveAbsJ jHomePos\NoEOffs,VSpeed,fine,tool0;
        ELSEIF bTopsy=TRUE AND bTurvey=FALSE THEN
            MoveAbsJ jTop1,VSpeed,fine,tDong;
            MoveAbsJ jTop2,VSpeed,fine,tDong;
            MoveJ Top3,vSpeed,z50,tDong;
            MoveJ Top4,vSpeed,fine,tDong;
            answer:=UIMessageBox(\Header:="What Are You Doing Step IRB-120"\MsgArray:=DTFTopMessage\BtnArray:=DTFTopButtons\Icon:=IconWarning);
            IF answer=1 THEN
                TPErase;
                TPwrite "OOH that Feels Nice";
                WHILE NThrustLoop>NCurrentThrustLoop DO

                    IF NCurrentThrustLoop=NThrustTemp2 THEN
                        TPwrite "HARDER DADDY";
                    ENDIF

                    IF NCurrentThrustLoop=NThrustTemp3 THEN
                        TPwrite "HARDER";
                    ENDIF

                    IF NCurrentThrustLoop=NThrustTemp4 THEN
                        TPwrite "HARDER";
                    ENDIF

                    IF NCurrentThrustLoop=NThrustTemp5 THEN
                        TPwrite "DONT STOP";
                    ENDIF

                    WHILE NCurrentThrustLoop>NThrustTemp5 AND NCurrentThrustLoop<=NThrustLoop DO
                        IF NCurrentThrustLoop=NThrustTemp5 THEN
                            TPwrite "OOH GOD YES";
                        ENDIF


                        IF NCurrentThrustLoop=NThrustTemp6 THEN
                            TPwrite "ALMOST THERE";
                        ENDIF

                        MoveL offs(Top4,0,0,-100),VSpeed,fine,tDong;
                        MoveL offs(Top4,0,0,-25),VSpeed,fine,tDong;

                        IF NCurrentThrustLoop=NThrustTemp7 THEN
                            TPwrite "BEEP BOP BOOP ---COMPLETION ACHIEVED---";
                            MoveL offs(Top4,0,5,-25),VSpeed,fine,tDong;
                            MoveL offs(Top4,0,0,-25),VSpeed,fine,tDong;
                            MoveL offs(Top4,0,5,-25),VSpeed,fine,tDong;
                            MoveL offs(Top4,0,0,-25),VSpeed,fine,tDong;
                            WaitTime .5;
                            MoveL offs(Top4,0,5,-25),VSpeed,fine,tDong;
                            MoveL offs(Top4,0,0,-25),VSpeed,fine,tDong;
                            MoveL offs(Top4,0,5,-25),VSpeed,fine,tDong;
                            MoveL offs(Top4,0,0,-25),VSpeed,fine,tDong;
                            WaitTime 5;
                        ENDIF

                        Incr NCurrentThrustLoop;
                    ENDWHILE
                    WaitTime 2;
                    Incr NCurrentThrustLoop;

                ENDWHILE
                answer:=UIMessageBox(\Header:="Was it good for you"\MsgArray:=DTFCompletionMessage\BtnArray:=DTFCompletionButtons\Icon:=IconWarning);
                IF answer=1 THEN
                ENDIF
                MoveL Top4,vSpeed,fine,tDong;
                MoveL Top3,vSpeed,z50,tDong;
                MoveAbsJ jTop2,VSpeed,fine,tDong;
                MoveAbsJ jTop1,VSpeed,fine,tDong;
            ELSEIF answer=2 THEN
                MoveAbsJ jTop1,VSpeed,fine,tool0;
            ENDIF
        ENDIF

    ENDPROC

!!!!!!!!!!!!!!!!!!!!!!!!!!!!!!!!!!!!!!!!!!!!!!!!!!!!!!!!!!!!!!!!!!!!!!!!!!!!!!!!!!!!!!!!!!!!!!!!!!

    PROC R_Docking_Menu()
        VAR num nMenuOption;
        VAR btnres btnresMainMenu;
        CONST Listitem ListOptions{7}:=[
        ["1","Select an option and press OK to run program"],
        ["2","Press CANCEL to return to Main Menu"],
        [""," "],
        [""," "],
        ["","SET SPEED"],
        ["","SET LOOP"],
        ["","RUN PROGRAM"]];

        !Menu Start
        bMenu:=True;
        WHILE bMenu DO
            nMenuOption:=UIListView(\Result:=btnresMainMenu\Header:="RUN DANCING QUEEN",ListOptions\Buttons:=btnOKCancel\Icon:=iconWarning);
            IF btnresMainMenu=resCancel Main_Menu;
            TEST nMenuOption
            CASE 1:
                TPErase;
                TPwrite "Wrong hole...WRONG HOLE!!!!!";
                waittime 5;
                TPErase;
            CASE 2:
                TPErase;
                TPwrite "Wrong hole...WRONG HOLE!!!!!";
                waittime 5;
                TPErase;
                RETURN ;
            CASE 3:
            CASE 4:
            CASE 5:
                R_Set_SPEEEEEED;
                R_Docking_Menu;
            CASE 6:
                NThrustLoop:=UINumEntry(\Header:="Set Repeat Counter"\MsgArray:=LoopMessage\Icon:=iconInfo\InitValue:=NThrustLoop\MinValue:=0\MaxValue:=1000);
                R_Docking_Menu;
            CASE 7:
                answer:=UIMessageBox(\Header:="CAUTION: ROBOT MAY MOVE"\MsgArray:=CautionMessage\BtnArray:=RunCancel\Icon:=IconWarning);
                IF answer=1 THEN
                    NCurrentThrustLoop:=0;
                    R_Docking;
                ELSEIF answer=2 THEN
                    RETURN ;
                ENDIF
                Main_Menu;
                bMenu:=False;
            ENDTEST
        ENDWHILE
    ENDPROC

    PROC R_Docking()
        CONST jointtarget j1:=[[0,0,-90,0,0,0],[9E+09,9E+09,9E+09,9E+09,9E+09,9E+09]];
        CONST jointtarget j2:=[[45,-34.7368,0,30,-45,0],[9E+09,9E+09,9E+09,9E+09,9E+09,9E+09]];
        CONST jointtarget j3:=[[-45,-35,0,-30,-45,0],[9E+09,9E+09,9E+09,9E+09,9E+09,9E+09]];
        CONST jointtarget j4:=[[45,-33.512,43.8106,8.56333E-05,-10.2984,-8.82129E-05],[9E+09,9E+09,9E+09,9E+09,9E+09,9E+09]];
        CONST jointtarget j5:=[[45,29.6234,-17.5512,3.19074E-05,-12.0721,-3.12018E-05],[9E+09,9E+09,9E+09,9E+09,9E+09,9E+09]];
        CONST jointtarget j6:=[[-45,-33.4907,43.6889,-7.08038E-05,-10.2336,-0.320042],[9E+09,9E+09,9E+09,9E+09,9E+09,9E+09]];
        CONST jointtarget j7:=[[-45,29.6402,-17.6857,-5.55671E-05,-11.99,-0.320058],[9E+09,9E+09,9E+09,9E+09,9E+09,9E+09]];
        CONST jointtarget j8:=[[45,19.6394,40.4538,2.45022E-06,-60.0932,-1.22166E-06],[9E+09,9E+09,9E+09,9E+09,9E+09,9E+09]];
        CONST jointtarget j9:=[[-45,19.6394,40.4538,2.45022E-06,-60.0932,-1.22166E-06],[9E+09,9E+09,9E+09,9E+09,9E+09,9E+09]];
        CONST jointtarget j10:=[[45,0,0,0,0,0],[9E+09,9E+09,9E+09,9E+09,9E+09,9E+09]];
        CONST jointtarget j11:=[[45,0,0,0,0,0],[9E+09,9E+09,9E+09,9E+09,9E+09,9E+09]];
        CONST jointtarget j12:=[[45,0,0,0,0,0],[9E+09,9E+09,9E+09,9E+09,9E+09,9E+09]];
        CONST jointtarget j13:=[[45,0,0,0,0,0],[9E+09,9E+09,9E+09,9E+09,9E+09,9E+09]];
        CONST jointtarget j14:=[[45,0,0,0,0,0],[9E+09,9E+09,9E+09,9E+09,9E+09,9E+09]];
        CONST jointtarget j15:=[[45,0,0,0,0,0],[9E+09,9E+09,9E+09,9E+09,9E+09,9E+09]];
        CONST jointtarget j16:=[[45,0,0,0,0,0],[9E+09,9E+09,9E+09,9E+09,9E+09,9E+09]];
        CONST jointtarget j17:=[[45,0,0,0,0,0],[9E+09,9E+09,9E+09,9E+09,9E+09,9E+09]];
        CONST jointtarget j18:=[[45,0,0,0,0,0],[9E+09,9E+09,9E+09,9E+09,9E+09,9E+09]];
        CONST jointtarget j19:=[[45,0,0,0,0,0],[9E+09,9E+09,9E+09,9E+09,9E+09,9E+09]];
        CONST jointtarget j20:=[[45,0,0,0,0,0],[9E+09,9E+09,9E+09,9E+09,9E+09,9E+09]];


        MoveAbsJ j1,VSpeed,fine,tool0;
        MoveAbsJ j2,VSpeed,fine,tool0;
        MoveAbsJ j1,VSpeed,fine,tool0;
        MoveAbsJ j2,VSpeed,fine,tool0;
        MoveAbsJ j1,VSpeed,fine,tool0;
        MoveAbsJ j3,VSpeed,fine,tool0;
        MoveAbsJ j1,VSpeed,fine,tool0;
        MoveAbsJ j3,VSpeed,fine,tool0;
        MoveAbsJ j1,VSpeed,fine,tool0;
        MoveAbsJ j4,VSpeed,fine,tool0;
        MoveAbsJ j1,VSpeed,fine,tool0;
        MoveAbsJ j4,VSpeed,fine,tool0;
        MoveAbsJ j1,VSpeed,fine,tool0;
        MoveAbsJ j5,VSpeed,fine,tool0;
        MoveAbsJ j1,VSpeed,fine,tool0;
        MoveAbsJ j5,VSpeed,fine,tool0;
        MoveAbsJ j1,VSpeed,fine,tool0;
        MoveAbsJ j6,VSpeed,fine,tool0;
        MoveAbsJ j1,VSpeed,fine,tool0;
        MoveAbsJ j6,VSpeed,fine,tool0;
        MoveAbsJ j1,VSpeed,fine,tool0;
        MoveAbsJ j7,VSpeed,fine,tool0;
        MoveAbsJ j1,VSpeed,fine,tool0;
        MoveAbsJ j7,VSpeed,fine,tool0;
        MoveAbsJ j1,VSpeed,fine,tool0;
        MoveAbsJ j8,VSpeed,fine,tool0;
        MoveAbsJ j1,VSpeed,fine,tool0;
        MoveAbsJ j8,VSpeed,fine,tool0;
        MoveAbsJ j1,VSpeed,fine,tool0;
        MoveAbsJ j9,VSpeed,fine,tool0;
        MoveAbsJ j1,VSpeed,fine,tool0;
        MoveAbsJ j9,VSpeed,fine,tool0;
        MoveAbsJ j8,VSpeed,fine,tool0;
        MoveAbsJ j9,VSpeed,fine,tool0;
        MoveAbsJ j8,VSpeed,fine,tool0;
        MoveAbsJ j9,VSpeed,fine,tool0;
        MoveAbsJ j6,VSpeed,fine,tool0;
        MoveAbsJ j7,VSpeed,fine,tool0;
        MoveAbsJ j6,VSpeed,fine,tool0;
        MoveAbsJ j7,VSpeed,fine,tool0;
        MoveAbsJ j6,VSpeed,fine,tool0;
        MoveAbsJ j4,VSpeed,fine,tool0;
        MoveAbsJ j5,VSpeed,fine,tool0;
        MoveAbsJ j4,VSpeed,fine,tool0;
        MoveAbsJ j5,VSpeed,fine,tool0;
        MoveAbsJ j4,VSpeed,fine,tool0;
        MoveAbsJ j2,VSpeed,fine,tool0;
        MoveAbsJ j3,VSpeed,fine,tool0;
        MoveAbsJ j2,VSpeed,fine,tool0;
        MoveAbsJ j3,VSpeed,fine,tool0;
        MoveAbsJ j1,VSpeed,fine,tool0;
        Incr NCurrentThrustLoop;
        IF NThrustLoop=0 OR NThrustLoop>NCurrentThrustLoop THEN
            R_Docking;
        ENDIF
        MoveAbsJ jHomePos\NoEOffs,VSpeed,fine,tool0;
        !Place Code Here
    ENDPROC

    !!!!!!!!!!!!!!!!!!!!!!!!!!!!!!!!!!!!!!!!!!!!!!!!!!!!!!!!!!!!!!!!!!

ENDMODULE

--- Backups/120-501650_Turvey/RAPID/TASK1/PROGMOD/M_Helicopter.mod ---
MODULE M_Helicopter
    !    !*****************************************************
    !    !Module Name:   M_TEMPLATE
    !    !Version:       1.22
    !    !Description:   Helicopter
    !    !Date:          2024-08-30
    !    !Author:        @ManicZanic
    !    !
    !    !*****************************************************
    !    !Change Log:
    !    !2024-08-31:    @ManicZanic - Orignal core pulled from MainModule
    !    !*****************************************************

    !HELICOPTER LOOP SWITCH
    PERS num nHelicopter:=1;

    PROC R_Helicopter_Menu()
        VAR num nMenuOption;
        VAR btnres btnresMainMenu;
        CONST Listitem ListOptions{7}:=[
        ["1","Select an option and press OK to run program"],
        ["2","Press CANCEL to return to Main Menu"],
        ["3"," "],
        ["4"," "],
        ["5","Set Speed"],
        ["6"," "],
        ["7","RUN PROGRAM"]];

        !       Menu Start
        bMenu:=True;
        WHILE bMenu DO
            nMenuOption:=UIListView(\Result:=btnresMainMenu\Header:="RUN Helicopter PROGRAM",ListOptions\Buttons:=btnOKCancel\Icon:=iconWarning);
            IF btnresMainMenu=resCancel Main_Menu;
            TEST nMenuOption
            CASE 1:
                TPErase;
                TPwrite "Wrong hole...WRONG HOLE!!!!!";
                waittime 5;
                TPErase;
            CASE 2:
                TPErase;
                TPwrite "Wrong hole...WRONG HOLE!!!!!";
                waittime 5;
                TPErase;
                Main_Menu;
            CASE 3:
            CASE 4:
            CASE 5:
                R_Set_SPEEEEEED;
                R_Helicopter_Menu;
            CASE 6:
            CASE 7:
                IF CondomMode=TRUE THEN
                    answer:=UIMessageBox(\Header:="CAUTION: ROBOT MAY MOVE"\MsgArray:=CautionMessage\BtnArray:=RunCancel\Icon:=IconWarning);
                    IF answer=1 THEN
                        NCameraLoop:=2;
                        R_Helicopter;
                        Main_Menu;
                    ELSEIF answer=2 THEN
                        Main_Menu;
                    ENDIF
                ELSE
                    NCameraLoop:=2;
                    R_Helicopter;
                    Main_Menu;
                ENDIF
                Main_Menu;
                bMenu:=False;
            ENDTEST
        ENDWHILE
    ENDPROC

    PROC R_Helicopter()
        CONST jointtarget jHelicopter:=[[0,26.8166,-4.77057,0,-22.0461,0],[9E+09,9E+09,9E+09,9E+09,9E+09,9E+09]];
        CONST robtarget H1:=[[640.50,-10,455.00],[0.707107,3.47691E-8,0.707107,-1.5478E-9],[-1,-1,0,1],[9E+9,9E+9,9E+9,9E+9,9E+9,9E+9]];
        CONST robtarget H2:=[[640.50,-10,440.00],[0.707107,7.61395E-9,0.707107,7.08051E-9],[-1,-1,0,1],[9E+9,9E+9,9E+9,9E+9,9E+9,9E+9]];
        CONST robtarget H3:=[[640.50,5,440.00],[0.707107,-7.61395E-9,0.707107,-7.08051E-9],[0,0,-1,1],[9E+9,9E+9,9E+9,9E+9,9E+9,9E+9]];
        CONST robtarget H4:=[[640.50,5,455.00],[0.707107,-3.47691E-8,0.707107,1.5478E-9],[0,0,-1,1],[9E+9,9E+9,9E+9,9E+9,9E+9,9E+9]];
        VAR num change_speed:=60;

        VSpeed:=V300;
        SpeedRefresh change_speed;
        IF NCameraLoop=2 THEN
            MoveAbsJ jHelicopter,v500,fine,tMain;
            NCameraLoop:=1;
        ENDIF
        MoveL H1,vSpeed,z50,tMain;
        MoveL H2,vSpeed,z50,tMain;
        MoveL H3,vSpeed,z50,tMain;
        MoveL H4,vSpeed,z50,tMain;
        R_Helicopter;
    ENDPROC
ENDMODULE

--- Backups/120-501650_Turvey/RAPID/TASK1/PROGMOD/M_TEMP.mod ---
MODULE M_TEMP
    !    !*****************************************************
    !    !Module Name:   M_TEMPLATE
    !    !Version:       1.22
    !    !Description:   Temp
    !    !Date:          2024-08-30
    !    !Author:        @ManicZanic
    !    !
    !    !*****************************************************
    !    !Change Log:
    !    !2024-08-31:    @ManicZanic - Orignal core pulled from MainModule
    !    !*****************************************************

    PROC Temp()

        CONST listitem list{3}:=[["","Item 1"],["","Item 2"],["","Item 3"]];
        VAR num list_item;
        VAR btnres button_answer;

        list_item:=UIListView(\Result:=button_answer\Header:="UIListView Header",list\Buttons:=btnOKCancel\Icon:=iconInfo\DefaultIndex:=1);
        IF button_answer=resOK THEN
            IF list_item=1 THEN
                ! Do item1
            ELSEIF list_item=2 THEN
                ! Do item 2
            ELSE
                ! Do item3
            ENDIF
        ELSE
            ! User has select Cancel
        ENDIF

    ENDPROC

ENDMODULE

--- Backups/120-501650_Turvey/RAPID/TASK1/PROGMOD/M_Template.mod ---
MODULE M_Template
    !    !*****************************************************
    !    !Module Name:   M_TEMPLATE
    !    !Version:       1.22
    !    !Description:   Program Template
    !    !Date:          2024-08-22
    !    !Author:        @ManicZanic
    !    !
    !    !*****************************************************
    !    !Change Log:
    !    !2024-08-22:    @ManicZanic - Orignal core structure developed
    !    !                           - Added Task specific Bool data
    !    !2024-08-22:    @ManicZanic - Set VersionID to match other modules
    !    !*****************************************************

    LOCAL PERS bool bTemplateMenu:=TRUE;
    CONST jointtarget jTemplatePos:=[[0,0,0,0,0,0],[9E+09,9E+09,9E+09,9E+09,9E+09,9E+09]];

    PROC R_Template_Menu()
        VAR num nMenuOption;!sets menu options
        VAR btnres btnresMainMenu;!Records button value

        !Sets the number of selectable items shown in the list view. Increasing / decreasing the number within {} will allow you to increase or decrease the number of options shown in the list
        CONST Listitem ListOptions{7}:=[["","Case 1 description"],["","Case 2 description"],["","Case 3 description"],["","Case 4 description"],["","Case 5 description"],["","Case 6 description"],["","Case 7 description"]];

        bTemplateMenu:=True;
        WHILE bTemplateMenu DO
            nMenuOption:=UIListView(\Result:=btnresMainMenu\Header:="Enter Header Here",ListOptions\Buttons:=btnOKCancel\Icon:=iconInfo);
            IF btnresMainMenu=resCancel return ;!When Cancel button pressed this returns you to previous menu
            TEST nMenuOption
            CASE 1:
                !Place Code for List item 1 here
                !Multiple calls can be made in a single case
                !If progam is large it is recommended to create a separate template
                !MoveAbsJ jTemplatePos,v500,fine,tool0; !Will move the robot to the template home position
                !R_Template !Will call the R_Template Procedure
                !RETURN; instruction will return to this menu once task is complete
            CASE 2:
                !Place Code for List item 2 here
            CASE 3:
                !Place Code for List item 3 here
            CASE 4:
                !Place Code for List item 4 here
            CASE 5:
                !Place Code for List item 5 here
            CASE 6:
                !Place Code for List item 6 here
            CASE 7:
                !Place Code for List item 7 here
                bTemplateMenu:=False;
            ENDTEST
        ENDWHILE
        bTemplateMenu:=True;
    ENDPROC

PROC R_Template()
    !PLACE CODE HERE
ENDPROC



ENDMODULE

--- Backups/120-501650_Turvey/RAPID/TASK1/PROGMOD/M_Tower_Of_Hanoi.mod ---
MODULE M_Tower_Of_Hanoi
    !    !*****************************************************
    !    !Module Name:   M_Tower_Of_Hanoi
    !    !Version:       1.22
    !    !Description:   Robot program to solve Tower of Haanoi
    !    !Date:          2024-08-01
    !    !Author:        @ManicZanic
    !    !               @ELIICE
    !    !               @Austin
    !    !*****************************************************
    !    !Change Log:
    !    !2024-08-01:    @ManicZanic - Orignal core structure developed
    !    !2024-08-01:    @ELIICE - Added to RobotStudio station and updated to function with graphics and added notes.
    !    !                       - Added additional variables for Movements.
    !    !                       - Added Initialize routine to automaticly reset working data variables.
    !    !                       - Reduced solution to the least number of Moves.
    !    !                       - Added General gripper IO signals. Control and state feedback.
    !    !2024-08-04:    @ManicZanic - Generated russan nesting doll style program to handle NOD values up to 10 discs.
    !    !                           - Added step count variables.
    !    !                           - Moved NOD selection to R_Shaft_Stroke_Test routine for easier counter selection.
    !    !2024-08-14:    @Austin - Added basic recursive solution to ToH problem (R_Recursive_Tower_Solution)
    !    !2024-08-21:    @ManicZanic - Added Menu options
    !    !                           - Moved non TOH routines to Main module.
    !    !                           - Reintegrated Recursive Solution into TOH module.
    !    !                           - Upgraded the speed selection menu
    !    !                           - Fromatted text
    !    !2024-08-22:    @ManicZanic - Removed unused code
    !    !                           - Added bTOHmenu bool data
    !    !2024-08-23:    @ManicZanic - Commented out parameters to maybe use later
    !    !2024-08-26:    @ManicZanic - Moved Speed to main
    !    !*****************************************************

    PERS tooldata tGripperTool:=[TRUE,[[0.000145392,0,140.499655058],[1,0,-0.000000126,0]],[1,[0,0,75],[1,0,0,0],0,0,0]];
    TASK PERS wobjdata wobjTower:=[FALSE,TRUE,"",[[0,600,150],[0.707106781,0,0,0.707106781]],[[0,0,0],[1,0,0,0]]];
    TASK PERS wobjdata wobjTower1:=[FALSE,TRUE,"",[[600,0,150],[1,0,0,0]],[[0,0,0],[1,0,0,0]]];
    LOCAL PERS bool bTOHMenu:=TRUE;

    !TOWER OF HANOI VARIABLES
    PERS num NDH:=6.35;!NOMINAL DISK HEIGHT
    PERS num NDD:=40;!NOMINAL DISK DIAMETER
    PERS num NSL:=65;!NOMINAL SHAFT LENGTH
    PERS num GOFz:=25;!GripperOffset
    PERS num GSafe:=75;!GripperSafeHeight
    PERS num NOD:=3;!NUMBER OF STACKED DISCS
    PERS num NStart:=2;!START POSITION
    PERS num NEnd:=3;!END POSITION
    PERS num NLoop:=1;!LOOP COUNT
    PERS num NMotionActive:=1;!0 ENABLES ROBOT MoveMENT WHILE 1 DISABLES ROBOT MoveMENT
    PERS num NStepCount:=11;!COMPLETED STEP COUNTER
    PERS num NtenDisc_Count:=26243;!TOTAL NUMBER OF CYCLES TO COMPLETE A 10 DISC TOWER IN STANDARD MODE.
    PERS num NJob:=4;!JOB SELECTION
    VAR num NFooBar:=0;!TEMP VAR FOR CALLING FUNC'S

    !WORKING DATA
    PERS num NShaft1X1:=-20;
    PERS num NShaft1Z1:=165;
    PERS num NShaft1Z2:=61.825;
    PERS num NShaft1Z3:=58.65;
    PERS num NShaft1Z4:=-25;
    PERS num NShaft2X1:=-20;
    PERS num NShaft2Z1:=165;
    PERS num NShaft2Z2:=61.825;
    PERS num NShaft2Z3:=58.65;
    PERS num NShaft2Z4:=0;
    PERS num NShaft3X1:=-20;
    PERS num NShaft3Z1:=165;
    PERS num NShaft3Z2:=61.825;
    PERS num NShaft3Z3:=58.65;
    PERS num NShaft3Z4:=19.05;


    CONST robtarget Shaft1:=[[0,200,0],[0.707106781,0,0.707106781,0],[0,0,-1,1],[9E+09,9E+09,9E+09,9E+09,9E+09,9E+09]];
    CONST robtarget Shaft2:=[[0,0,0],[0.707106781,0,0.707106781,0],[0,0,0,1],[9E+09,9E+09,9E+09,9E+09,9E+09,9E+09]];
    CONST robtarget Shaft3:=[[0,-200,0],[0.707106781,0,0.707106781,0],[-1,-1,0,1],[9E+09,9E+09,9E+09,9E+09,9E+09,9E+09]];

    PROC R_Tower_Of_Hanoi_Menu()
        VAR num nMenuOption;
        VAR btnres btnresMainMenu;
        CONST Listitem ListOptions{7}:=[["","Run Program"],["","Set Number of Discs"],["","Set Nominal Disc Dimension"],["","Set Nominal Disc Height"],["","Set Nominal Shaft Length"],["","Set Speed"],["","Activate / Deactivate Motion"]];

        bTOHMenu:=True;
        WHILE bTOHMenu DO
            nMenuOption:=UIListView(\Result:=btnresMainMenu\Header:="Tower Of Hanoi MAIN MENU",ListOptions\Buttons:=btnOKCancel\Icon:=iconInfo);
            IF btnresMainMenu=resCancel return ;
            TEST nMenuOption
            CASE 1:
                R_Tower_Of_Hanoi_SolSel;
            CASE 2:
                NOD:=UINumEntry(\Header:="Update Number Of Discs"\Message:="Enter Number Of Stacked Discs"\Icon:=iconInfo\InitValue:=NOD\MinValue:=0\MaxValue:=10);
                R_Tower_Of_Hanoi_Menu;
            CASE 3:
                NDD:=UINumEntry(\Header:="Update Nominal Disc Diameter (Metric)"\Message:="Enter Nominal Disc Diameter (mm) Of Largest Dics In The Stack"\Icon:=iconInfo\InitValue:=NDD\MinValue:=0\MaxValue:=1000);
                R_Tower_Of_Hanoi_Menu;
            CASE 4:
                NDH:=UINumEntry(\Header:="Update Nominal Disc Height (Metric)"\Message:="Enter Nominal Disc Height (mm)"\Icon:=iconInfo\InitValue:=NDH\MinValue:=0\MaxValue:=100);
                R_Tower_Of_Hanoi_Menu;
            CASE 5:
                NSL:=UINumEntry(\Header:="Update Nominal Shaft Length (Metric)"\Message:="Enter Nominal Shaft Length (mm)"\Icon:=iconInfo\InitValue:=NSL\MinValue:=0\MaxValue:=2000);
                R_Tower_Of_Hanoi_Menu;
            CASE 6:
                R_Set_SPEEEEEED;
                R_Tower_Of_Hanoi_Menu;
            CASE 7:
                NMotionActive:=UINumEntry(\Header:="Motion Activation"\Message:="Enter 1 to Enable Motion Enter 0 to Disable Motion"\Icon:=iconInfo\InitValue:=NMotionActive\MinValue:=0\MaxValue:=1);
                R_Tower_Of_Hanoi_Menu;
                bTOHMenu:=False;
            ENDTEST
        ENDWHILE
        bTOHMenu:=True;
    ENDPROC

    FUNC num R_Recursive_Tower_Solution(num NCounter,num NFromRod,num NToRod,num NAuxRod)
        !Modeled after https://www.geeksforgeeks.org/c-program-for-tower-of-hanoi/
        IF NCounter=0 THEN
            RETURN 0;
        ENDIF
        NFooBar:=R_Recursive_Tower_Solution(NCounter-1,NFromRod,NAuxRod,NToRod);
        TPWrite "Disk to move: "\Num:=NCounter;
        TPWrite "Source rod: "\Num:=NFromRod;
        TPWrite "Destination Rod: "\Num:=NToRod;
        TPWrite "Moving...";
        NStart:=NFromRod;
        NEnd:=NToRod;
        R_Pick_N_Place;
        TPWrite "Move complete. Onto next move...";
        TPWrite "****************************************";
        NFooBar:=R_Recursive_Tower_Solution(NCounter-1,NAuxRod,NToRod,NFromRod);
        RETURN 0;
    ENDFUNC

    PROC R_Tower_Of_Hanoi_SolSel()
        VAR num nMenuOption;
        VAR btnres btnresMainMenu;
        CONST Listitem ListOptions{7}:=[["","Select solution method and press OK to run program"],["","Press CANCEL to return to previous menu"],[""," "],[""," "],[""," "],["","STANDARD"],["","RECURSION"]];

        bTOHMenu:=True;
        WHILE bTOHMenu DO
            nMenuOption:=UIListView(\Result:=btnresMainMenu\Header:="Tower Of Hanoi PROGRAM MENU",ListOptions\Buttons:=btnOKCancel\Icon:=iconWarning);
            IF btnresMainMenu=resCancel return ;
            TEST nMenuOption
            CASE 1:
                TPErase;
                TPwrite "Wrong hole...WRONG HOLE!!!!!";
                waittime 5;
                TPErase;
            CASE 2:
                TPErase;
                TPwrite "Wrong hole...WRONG HOLE!!!!!";
                waittime 5;
                TPErase;
                R_Tower_Of_Hanoi_SolSel;
            CASE 3:
            CASE 4:
            CASE 5:
                R_Set_SPEEEEEED;
                R_Tower_Of_Hanoi_SolSel;
            CASE 6:
            answer:= UIMessageBox ( \Header:="CAUTION: ROBOT MAY MOVE" \MsgArray:=CautionMessage \BtnArray:=RunCancel \Icon:=IconWarning);
            IF answer = 1 THEN
                Initialize;
                R_Tower_Of_Hanoi;
            ELSEIF answer = 2 THEN
                Main;
            ENDIF
                Main;
            CASE 7:
            answer:= UIMessageBox ( \Header:="CAUTION: ROBOT MAY MOVE" \MsgArray:=CautionMessage \BtnArray:=RunCancel \Icon:=IconWarning);
            IF answer = 1 THEN
                Initialize;
                NFooBar:=R_Recursive_Tower_Solution(NOD,1,3,2);!Moving from rod 1 to rod 3, rod 2 is aux;
            ELSEIF answer = 2 THEN
                Main;
            ENDIF
                Main;
                bTOHMenu:=False;
            ENDTEST
        ENDWHILE
        bTOHMenu:=True;
    ENDPROC

    PROC Initialize()
        !Reset Grippers I/O and sequence communication bits

        !SHAFT 1 WORKING DATA

        !Shaft Approach Side.
        NShaft1X1:=-(NDD/2);
        !Shaft Approach Above. Calculate from values to clear the shaft holding disk
        NShaft1Z1:=NSL+GOFz+GSafe;
        !Shaft Drop Position Start
        NShaft1Z2:=NSL-(NDH/2);
        !Shaft Drop Position End
        NShaft1Z3:=NSL-(NDH);
        !Shaft Pick Position. Reset to zero.
        NShaft1Z4:=-0;

        !SHAFT 2 WORKING DATA
        !Shaft Approach Side.
        NShaft2X1:=-(NDD/2);
        !Shaft Approach Above. Calculate from values to clear the shaft holding disk
        NShaft2Z1:=NSL+GOFz+GSafe;
        !Shaft Drop Position Start
        NShaft2Z2:=NSL-(NDH/2);
        !Shaft Drop Position End
        NShaft2Z3:=NSL-(NDH);
        !Shaft Pick Position. Reset to zero.
        NShaft2Z4:=-0;

        !SHAFT 3  WORKING DATA
        !Shaft Approach Side.
        NShaft3X1:=-(NDD/2);
        !Shaft Approach Above. Calculate from values to clear the shaft holding disk
        NShaft3Z1:=NSL+GOFz+GSafe;
        !Shaft Drop Position Start
        NShaft3Z2:=NSL-(NDH/2);
        !Shaft Drop Position End
        NShaft3Z3:=NSL-(NDH);
        !Shaft Pick Position. Reset to zero.
        NShaft3Z4:=-0;

        !Calculate pick height
        !Number of Disks x Nominal Disk Height
        NShaft1Z4:=NOD*NDH-GOFz;
        NShaft2Z4:=(0);
        NShaft3Z4:=(0);

    ENDPROC

    PROC R_Handy()
        !The_Stroke_Handler
        !Modify the following positions to define the locations of each shaft
        MoveL Shaft1,v100,fine,tGripperTool;
        MoveL Shaft2,v100,fine,tGripperTool;
        MoveL Shaft3,v100,fine,tGripperTool;
    ENDPROC

    PROC R_Tower_Of_Hanoi()
        MoveAbsJ jHomePos,v500,fine,tGripperTool;
        NStepCount:=0;!Resets NStepCount to 0
        NLoop:=1;!Resets NLoop to 0
        NOD:=NOD;
        IF NOD=1 THEN
            R_Tier1;
        ENDIF
        IF NOD=2 THEN
            R_Tier2;
        ENDIF
        IF NOD=3 THEN
            R_Tier3;
        ENDIF
        IF NOD=4 THEN
            R_Tier4;
        ENDIF
        IF NOD=5 THEN
            R_Tier5;
        ENDIF
        IF NOD=6 THEN
            R_Tier6;
        ENDIF
        IF NOD=7 THEN
            R_Tier7;
        ENDIF
        IF NOD=8 THEN
            R_Tier8;
        ENDIF
        IF NOD=9 THEN
            R_Tier9;
        ENDIF
        IF NOD=10 THEN
            R_Tier10;
        ENDIF
        MoveAbsJ jHomePos,v500,fine,tool0;
        !Puzzle solved reset values and stop
        !        StopMoveReset\AllMotionTasks;
    ENDPROC

    PROC R_Pick_N_Place()
        IF NMotionActive=1 then
            if NStart=1 then
                MoveJ offs(Shaft1,NShaft1X1,0,NShaft1Z1),VSpeed,z5,tGripperTool\Wobj:=wobjTower;
                MoveL offs(Shaft1,NShaft1X1,0,NShaft1Z4),VSpeed,z5,tGripperTool\Wobj:=wobjTower;
                MoveL offs(Shaft1,0,0,NShaft1Z4),VSpeed,fine,tGripperTool\Wobj:=wobjTower;
                !CLOSE GRIPPER
                !PulseDO \PLength:=1, DO_GripperClose;
                WaitTime 0.2;
                !WaitDI DI_GripperClosed,1 \MaxTime:=0.5;
                MoveL offs(Shaft1,0,0,NShaft1Z1),VSpeed,z5,tGripperTool\Wobj:=wobjTower;
                NShaft1Z4:=NShaft1Z4-NDH;
            ENDIF
            if NStart=2 then
                MoveJ offs(Shaft2,NShaft2X1,0,NShaft2Z1),VSpeed,z5,tGripperTool\Wobj:=wobjTower;
                MoveL offs(Shaft2,NShaft2X1,0,NShaft2Z4),VSpeed,z5,tGripperTool\Wobj:=wobjTower;
                MoveL offs(Shaft2,0,0,NShaft2Z4),VSpeed,fine,tGripperTool\Wobj:=wobjTower;
                !CLOSE GRIPPER
                !PulseDO \PLength:=1, DO_GripperClose;
                WaitTime 0.2;
                !WaitDI DI_GripperClosed,1 \MaxTime:=0.5;
                MoveL offs(Shaft2,0,0,NShaft2Z1),VSpeed,z5,tGripperTool\Wobj:=wobjTower;
                NShaft2Z4:=NShaft2Z4-NDH;
            ENDIF
            if NStart=3 then
                MoveJ offs(Shaft3,NShaft3X1,0,NShaft3Z1),VSpeed,z5,tGripperTool\Wobj:=wobjTower;
                MoveL offs(Shaft3,NShaft3X1,0,NShaft3Z4),VSpeed,z5,tGripperTool\Wobj:=wobjTower;
                MoveL offs(Shaft3,0,0,NShaft3Z4),VSpeed,fine,tGripperTool\Wobj:=wobjTower;
                !CLOSE GRIPPER
                !PulseDO \PLength:=1, DO_GripperClose;
                WaitTime 0.2;
                !WaitDI DI_GripperClosed,1 \MaxTime:=0.5;
                MoveL offs(Shaft3,0,0,NShaft3Z1),VSpeed,z5,tGripperTool\Wobj:=wobjTower;
                NShaft3Z4:=NShaft3Z4-NDH;
            ENDIF
            if NEnd=1 then
                MoveJ offs(Shaft1,0,0,NShaft1Z1),VSpeed,z5,tGripperTool\Wobj:=wobjTower;
                MoveL offs(Shaft1,0,0,NShaft1Z2),VSpeed,fine,tGripperTool\Wobj:=wobjTower;
                !OPEN GRIPPER
                !PulseDO \Plength:=1,DO_GripperClose;
                WaitTime 0.2;
                !WaitDI DI_GripperOpened,1 \MaxTime:=0.5;
                MoveL offs(Shaft1,NShaft1X1,0,NShaft1Z3),VSpeed,z0,tGripperTool\Wobj:=wobjTower;
                MoveL offs(Shaft1,0,0,NShaft1Z1),VSpeed,z5,tGripperTool\Wobj:=wobjTower;
                NShaft1Z4:=NShaft1Z4+NDH;
            ENDIF
            if NEnd=2 THEN
                MoveJ offs(Shaft2,0,0,NShaft2Z1),VSpeed,z5,tGripperTool\Wobj:=wobjTower;
                MoveL offs(Shaft2,0,0,NShaft2Z2),VSpeed,fine,tGripperTool\Wobj:=wobjTower;
                !OPEN GRIPPER
                !PulseDO \Plength:=1,DO_GripperClose;
                WaitTime 0.2;
                !WaitDI DI_GripperOpened,1 \MaxTime:=0.5;
                MoveL offs(Shaft2,NShaft2X1,0,NShaft2Z3),VSpeed,z0,tGripperTool\Wobj:=wobjTower;
                MoveL offs(Shaft2,0,0,NShaft2Z1),VSpeed,z5,tGripperTool\Wobj:=wobjTower;
                NShaft2Z4:=NShaft2Z4+NDH;
            ENDIF
            IF NEnd=3 THEN
                MoveJ offs(Shaft3,0,0,NShaft3Z1),VSpeed,z5,tGripperTool\Wobj:=wobjTower;
                MoveL offs(Shaft3,0,0,NShaft3Z2),VSpeed,fine,tGripperTool\Wobj:=wobjTower;
                !OPEN GRIPPER
                !PulseDO \Plength:=1,DO_GripperClose;
                WaitTime 0.2;
                !WaitDI DI_GripperOpened,1 \MaxTime:=0.5;
                MoveL offs(Shaft3,NShaft3X1,0,NShaft3Z3),VSpeed,z0,tGripperTool\Wobj:=wobjTower;
                MoveL offs(Shaft3,0,0,NShaft3Z1),VSpeed,z5,tGripperTool\Wobj:=wobjTower;
                NShaft3Z4:=NShaft3Z4+NDH;
            ENDIF
        ENDIF
        incr NStepCount;
    ENDPROC

    PROC R_Tier1()
        IF NOD=1 THEN
            NStart:=1;
            NEnd:=3;
            R_Pick_N_Place;
        ENDIF
        IF NOD>1 THEN
            NStart:=1;
            NEnd:=2;
            R_Pick_N_Place;
        ENDIF
    ENDPROC

    PROC R_Tier2()
        IF NOD>=2 AND NLoop=1 THEN
            NStart:=1;
            NEnd:=2;
            R_Pick_N_Place;
            NStart:=1;
            NEnd:=3;
            R_Pick_N_Place;
            NStart:=2;
            NEnd:=3;
            R_Pick_N_Place;
        ENDIF
        IF NOD>2 AND NLoop=2 THEN
            NStart:=3;
            NEnd:=2;
            R_Pick_N_Place;
            NStart:=3;
            NEnd:=1;
            R_Pick_N_Place;
            NStart:=2;
            NEnd:=1;
            R_Pick_N_Place;
        ENDIF
    ENDPROC

    PROC R_Tier3()
        !Move tier 3 to the right tower
        IF NOD>=3 AND NLoop=1 THEN
            R_Tier2;
            NLoop:=2;
            NStart:=1;
            NEnd:=2;
            R_Pick_N_Place;
            R_Tier2;
            NLoop:=1;
            NStart:=2;
            NEnd:=3;
            R_Pick_N_Place;
            R_Tier2;
        ENDIF
        !Move tier 3 to the left tower
        IF NOD>3 AND NLoop=2 THEN
            R_Tier2;
            NLoop:=1;
            NStart:=3;
            NEnd:=2;
            R_Pick_N_Place;
            R_Tier2;
            NLoop:=2;
            NStart:=2;
            NEnd:=1;
            R_Pick_N_Place;
            R_Tier2;
        ENDIF
    ENDPROC

    PROC R_Tier4()
        !Move tier 4 to the right tower
        IF NOD>=4 AND NLoop=1 THEN
            R_Tier3;
            NLoop:=2;
            NStart:=1;
            NEnd:=2;
            R_Pick_N_Place;
            R_Tier3;
            NLoop:=1;
            NStart:=2;
            NEnd:=3;
            R_Pick_N_Place;
            R_Tier3;
        ENDIF
        !Move tier 4 to the left tower
        IF NOD>4 AND NLoop=2 THEN
            R_Tier3;
            NLoop:=1;
            NStart:=3;
            NEnd:=2;
            R_Pick_N_Place;
            R_Tier3;
            NLoop:=2;
            NStart:=2;
            NEnd:=1;
            R_Pick_N_Place;
            R_Tier3;
        ENDIF
    ENDPROC

    PROC R_Tier5()
        !Move tier 5 to the right tower
        IF NOD>=5 AND NLoop=1 THEN
            R_Tier4;
            NLoop:=2;
            NStart:=1;
            NEnd:=2;
            R_Pick_N_Place;
            R_Tier4;
            NLoop:=1;
            NStart:=2;
            NEnd:=3;
            R_Pick_N_Place;
            R_Tier4;
        ENDIF
        !Move tier 5 to the left tower
        IF NOD>5 AND NLoop=2 THEN
            R_Tier4;
            NLoop:=1;
            NStart:=3;
            NEnd:=2;
            R_Pick_N_Place;
            R_Tier4;
            NLoop:=2;
            NStart:=2;
            NEnd:=1;
            R_Pick_N_Place;
            R_Tier4;
        ENDIF
    ENDPROC

    PROC R_Tier6()
        !Move Tier 6 to the right tower
        IF NOD>=6 AND NLoop=1 THEN
            R_Tier5;
            NLoop:=2;
            NStart:=1;
            NEnd:=2;
            R_Pick_N_Place;
            R_Tier5;
            NLoop:=1;
            NStart:=2;
            NEnd:=3;
            R_Pick_N_Place;
            R_Tier5;
        ENDIF
        !Move Tier 6 to the left tower
        IF NOD>6 AND NLoop=2 THEN
            R_Tier5;
            NLoop:=1;
            NStart:=3;
            NEnd:=2;
            R_Pick_N_Place;
            R_Tier5;
            NLoop:=2;
            NStart:=2;
            NEnd:=1;
            R_Pick_N_Place;
            R_Tier5;
        ENDIF
    ENDPROC

    PROC R_Tier7()
        !Move Tier 7 to the right tower
        IF NOD>=7 AND NLoop=1 THEN
            R_Tier6;
            NLoop:=2;
            NStart:=1;
            NEnd:=2;
            R_Pick_N_Place;
            R_Tier6;
            NLoop:=1;
            NStart:=2;
            NEnd:=3;
            R_Pick_N_Place;
            R_Tier6;
        ENDIF
        !Move Tier 7 to the left tower
        IF NOD>7 AND NLoop=2 THEN
            R_Tier6;
            NLoop:=1;
            NStart:=3;
            NEnd:=2;
            R_Pick_N_Place;
            R_Tier6;
            NLoop:=2;
            NStart:=2;
            NEnd:=1;
            R_Pick_N_Place;
            R_Tier6;
        ENDIF
    ENDPROC

    PROC R_Tier8()
        !Move Tier 8 to the right tower
        IF NOD>=8 AND NLoop=1 THEN
            R_Tier7;
            NLoop:=2;
            NStart:=1;
            NEnd:=2;
            R_Pick_N_Place;
            R_Tier7;
            NLoop:=1;
            NStart:=2;
            NEnd:=3;
            R_Pick_N_Place;
            R_Tier7;
        ENDIF
        !Move Tier 8 to the left tower
        IF NOD>8 AND NLoop=2 THEN
            R_Tier7;
            NLoop:=1;
            NStart:=3;
            NEnd:=2;
            R_Pick_N_Place;
            R_Tier7;
            NLoop:=2;
            NStart:=2;
            NEnd:=1;
            R_Pick_N_Place;
            R_Tier7;
        ENDIF
    ENDPROC

    PROC R_Tier9()
        !Move Tier 9 to the right tower
        IF NOD>=9 AND NLoop=1 THEN
            R_Tier8;
            NLoop:=2;
            NStart:=1;
            NEnd:=2;
            R_Pick_N_Place;
            R_Tier8;
            NLoop:=1;
            NStart:=2;
            NEnd:=3;
            R_Pick_N_Place;
            R_Tier8;
        ENDIF
        !Move Tier 9 to the left tower
        IF NOD>9 AND NLoop=2 THEN
            R_Tier8;
            NLoop:=1;
            NStart:=3;
            NEnd:=2;
            R_Pick_N_Place;
            R_Tier8;
            NLoop:=2;
            NStart:=2;
            NEnd:=1;
            R_Pick_N_Place;
            R_Tier8;
        ENDIF
    ENDPROC

    PROC R_Tier10()
        !Move Tier 10 to the right tower
        IF NOD>=10 AND NLoop=1 THEN
            R_Tier9;
            NLoop:=2;
            NStart:=1;
            NEnd:=2;
            R_Pick_N_Place;
            R_Tier9;
            NLoop:=1;
            NStart:=2;
            NEnd:=3;
            R_Pick_N_Place;
            R_Tier9;
        ENDIF
        !Move Tier 10 to the left tower
        IF NOD>10 AND NLoop=2 THEN
            R_Tier9;
            NLoop:=1;
            NStart:=3;
            NEnd:=2;
            R_Pick_N_Place;
            R_Tier9;
            NLoop:=2;
            NStart:=2;
            NEnd:=1;
            R_Pick_N_Place;
            R_Tier9;
        ENDIF

    ENDPROC


ENDMODULE

--- Backups/120-501650_Turvey/RAPID/TASK1/PROGMOD/M_Yoga.mod ---
MODULE M_Yoga
    !    !*****************************************************
    !    !Module Name:   M_TEMPLATE
    !    !Version:       1.22
    !    !Description:   Yoga
    !    !Date:          2024-08-30
    !    !Author:        @ManicZanic
    !    !
    !    !*****************************************************
    !    !Change Log:
    !    !2024-08-31:    @ManicZanic - Orignal core pulled from MainModule
    !    !*****************************************************

        CONST jointtarget jCobra:=[[-45,-80,10,35,60,0],[9E+09,9E+09,9E+09,9E+09,9E+09,9E+09]];
        CONST jointtarget jDoggyStyle:=[[0,20,60,55,-55,0],[9E+09,9E+09,9E+09,9E+09,9E+09,9E+09]];
        CONST jointtarget jCamel:=[[0,50,-100,0,-60,0],[9E+09,9E+09,9E+09,9E+09,9E+09,9E+09]];
        CONST jointtarget jChair:=[[0,-70,60,0,80,0],[9E+09,9E+09,9E+09,9E+09,9E+09,9E+09]];
        CONST jointtarget jStarGazer:=[[0,0,-90,0,0,0],[9E+09,9E+09,9E+09,9E+09,9E+09,9E+09]];


    PROC R_YogaPose()
        VAR num nMenuOption;
        VAR btnres btnresMainMenu;
        CONST Listitem ListOptions{9}:=[
        ["1","Select an option and press OK to run program"],
        ["2","Press CANCEL to return to Main Menu"],
        ["3"," "],["4","Cobra"],
        ["5","Doggy Style"],
        ["6","Camel"],
        ["7","Chair"],
        ["8","Star Gazer"],
        ["9"," "]];

        !       Menu Start
        bMenu:=True;
        WHILE bMenu DO
            nMenuOption:=UIListView(\Result:=btnresMainMenu\Header:="SELECT YOGA POSE",ListOptions\Buttons:=btnOKCancel\Icon:=iconWarning);
            IF btnresMainMenu=resCancel Main_Menu;
            TEST nMenuOption
            CASE 1:
                TPErase;
                TPwrite "Wrong hole...WRONG HOLE!!!!!";
                waittime 5;
                TPErase;
            CASE 2:
                TPErase;
                TPwrite "Wrong hole...WRONG HOLE!!!!!";
                waittime 5;
                TPErase;
                RETURN ;
            CASE 3:
            CASE 4:
                IF CondomMode=TRUE THEN
                    answer:=UIMessageBox(\Header:="CAUTION: ROBOT MAY MOVE"\MsgArray:=CautionMessage\BtnArray:=RunCancel\Icon:=IconWarning);
                    IF answer=1 THEN
                        MoveAbsJ jCobra,v150,fine,tool0;
                    ELSEIF answer=2 THEN
                        RETURN ;
                    ENDIF
                ELSE
                    MoveAbsJ jCobra,v150,fine,tool0;
                ENDIF
                R_YogaPose;
            CASE 5:
                IF CondomMode=TRUE THEN
                    answer:=UIMessageBox(\Header:="CAUTION: ROBOT MAY MOVE"\MsgArray:=CautionMessage\BtnArray:=RunCancel\Icon:=IconWarning);
                    IF answer=1 THEN
                        MoveAbsJ jDoggyStyle,v150,fine,tool0;
                    ELSEIF answer=2 THEN
                        RETURN ;
                    ENDIF
                ELSE
                    MoveAbsJ jDoggyStyle,v150,fine,tool0;
                ENDIF
                R_YogaPose;
            CASE 6:
                IF CondomMode=TRUE THEN
                    answer:=UIMessageBox(\Header:="CAUTION: ROBOT MAY MOVE"\MsgArray:=CautionMessage\BtnArray:=RunCancel\Icon:=IconWarning);
                    IF answer=1 THEN
                        MoveAbsJ jCamel,v150,fine,tool0;
                    ELSEIF answer=2 THEN
                        RETURN ;
                    ENDIF
                ELSE
                    MoveAbsJ jCamel,v150,fine,tool0;
                ENDIF
                R_YogaPose;
            CASE 7:
                IF CondomMode=TRUE THEN
                    answer:=UIMessageBox(\Header:="CAUTION: ROBOT MAY MOVE"\MsgArray:=CautionMessage\BtnArray:=RunCancel\Icon:=IconWarning);
                    IF answer=1 THEN
                        MoveAbsJ jChair,v150,fine,tool0;
                    ELSEIF answer=2 THEN
                        RETURN ;
                    ENDIF
                ELSE
                    MoveAbsJ jChair,v150,fine,tool0;
                ENDIF
                R_YogaPose;
            CASE 8:
                IF CondomMode=TRUE THEN
                    answer:=UIMessageBox(\Header:="CAUTION: ROBOT MAY MOVE"\MsgArray:=CautionMessage\BtnArray:=RunCancel\Icon:=IconWarning);
                    IF answer=1 THEN
                        MoveAbsJ jStarGazer,v150,fine,tool0;
                    ELSEIF answer=2 THEN
                        RETURN ;
                    ENDIF
                ELSE
                    MoveAbsJ jStarGazer,v150,fine,tool0;
                    TPErase;
                    TPWrite "HEY LOOK A ROCKET SHIP";
                    WaitTime 2;
                    TPWrite "*      *      *";
                    TPWrite "*    *       *    *";
                    TPWrite "   8=====D~~...___";
                    TPWrite "*      *      *";
                    TPWrite "*    *       *    *";
                    WaitTime 5;
                    TPErase;
                    R_YogaPose;
                ENDIF
            CASE 9:
                bMenu:=False;
            ENDTEST
        ENDWHILE
    ENDPROC
ENDMODULE

--- Backups/120-501650_Turvey/SYSPAR/EIO.cfg ---
EIO:CFG_1.0:5:0::
#
EIO_BUS:

      -Name "Virtual1" -ConnectorID "SIM1"

      -Name "DeviceNet_Lean" -BusType "DNLE" -ConnectorID "PCI1"\
      -ConnectorLabel "DeviceNet Lean"
#
EIO_UNIT_TYPE:

      -Name "Virtual" -VendorName "ABB" -ProductName "Virtual unit"

      -Name "d651_Lean" -BusType "DNLE" -VendorName "ABB Robotics"\
      -ProductName "Combi Unit" -DL_ProductCode 25

      -Name "d652_Lean" -BusType "DNLE" -VendorName "ABB Robotics"\
      -ProductName "24 VDC Unit" -DL_ProductCode 26

      -Name "d653_Lean" -BusType "DNLE" -VendorName "ABB Robotics"\
      -ProductName "Relay Unit" -DL_ProductCode 27

      -Name "AC500_PLC_Lean" -BusType "DNLE" -VendorName "ABB Stotz"\
      -ProductName "AC500 PLC - FPB" -DL_ProductCode 1 -DL_VendorID 760

      -Name "DL_GENERIC" -BusType "DNLE" -DL_ProductCode 3535

      -Name "DL_GENERIC_POLL" -BusType "DNLE" -DL_ProductCode 3535\
      -DL_Pollrate 30

      -Name "d351_Lean" -BusType "DNLE" -VendorName "ABB Robotics"\
      -ProductName "IBS Adapter" -DL_ProductCode 7

      -Name "d352_Lean" -BusType "DNLE" -VendorName "ABB Robotics"\
      -ProductName "PBUS Adapter" -DL_ProductCode 8

      -Name "d378_Lean" -BusType "DNLE" -VendorName "ABB Robotics"\
      -ProductName "CCLink Adapter" -DL_ProductCode 17
#
EIO_UNIT:

      -Name "BOARD10" -UnitType "d652_Lean" -Bus "DeviceNet_Lean" -DL_Address 10
#
EIO_SIGNAL:

      -Name "DI10_1" -SignalType "DI" -Unit "BOARD10" -UnitMap "0"

      -Name "DI10_2" -SignalType "DI" -Unit "BOARD10" -UnitMap "1"

      -Name "DI10_3" -SignalType "DI" -Unit "BOARD10" -UnitMap "2"

      -Name "DI10_4" -SignalType "DI" -Unit "BOARD10" -UnitMap "3"

      -Name "DI10_5" -SignalType "DI" -Unit "BOARD10" -UnitMap "4"

      -Name "DI10_6" -SignalType "DI" -Unit "BOARD10" -UnitMap "5"

      -Name "DI10_7" -SignalType "DI" -Unit "BOARD10" -UnitMap "6"

      -Name "DI10_8" -SignalType "DI" -Unit "BOARD10" -UnitMap "7"

      -Name "DI10_9" -SignalType "DI" -Unit "BOARD10" -UnitMap "8"

      -Name "DI10_10" -SignalType "DI" -Unit "BOARD10" -UnitMap "9"

      -Name "DI10_11" -SignalType "DI" -Unit "BOARD10" -UnitMap "10"

      -Name "DI10_12" -SignalType "DI" -Unit "BOARD10" -UnitMap "11"

      -Name "DI10_13" -SignalType "DI" -Unit "BOARD10" -UnitMap "12"

      -Name "DI10_14" -SignalType "DI" -Unit "BOARD10" -UnitMap "13"

      -Name "DI10_15" -SignalType "DI" -Unit "BOARD10" -UnitMap "14"

      -Name "DI10_16" -SignalType "DI" -Unit "BOARD10" -UnitMap "15"

      -Name "DO10_1" -SignalType "DO" -Unit "BOARD10" -UnitMap "0"

      -Name "DO10_2" -SignalType "DO" -Unit "BOARD10" -UnitMap "1"

      -Name "DO10_3" -SignalType "DO" -Unit "BOARD10" -UnitMap "2"

      -Name "DO10_4" -SignalType "DO" -Unit "BOARD10" -UnitMap "3"

      -Name "DO10_5" -SignalType "DO" -Unit "BOARD10" -UnitMap "4"

      -Name "DO10_6" -SignalType "DO" -Unit "BOARD10" -UnitMap "5"

      -Name "DO10_7" -SignalType "DO" -Unit "BOARD10" -UnitMap "6"

      -Name "DO10_8" -SignalType "DO" -Unit "BOARD10" -UnitMap "7"

      -Name "DO10_9" -SignalType "DO" -Unit "BOARD10" -UnitMap "8"

      -Name "DO10_10" -SignalType "DO" -Unit "BOARD10" -UnitMap "9"

      -Name "DO10_11" -SignalType "DO" -Unit "BOARD10" -UnitMap "10"

      -Name "DO10_12" -SignalType "DO" -Unit "BOARD10" -UnitMap "11"

      -Name "DO10_13" -SignalType "DO" -Unit "BOARD10" -UnitMap "12"

      -Name "DO10_14" -SignalType "DO" -Unit "BOARD10" -UnitMap "13"

      -Name "DO10_15" -SignalType "DO" -Unit "BOARD10" -UnitMap "14"

      -Name "DO10_16" -SignalType "DO" -Unit "BOARD10" -UnitMap "15"

      -Name "SOManButt_On1" -SignalType "DO" -Unit "BOARD10" -UnitMap "41"\
      -Access "All" -SysfailReset

      -Name "SOManButt_On2" -SignalType "DO" -Unit "BOARD10" -UnitMap "42"\
      -Access "All" -SysfailReset

      -Name "SOManButt_On4" -SignalType "DO" -Unit "BOARD10" -UnitMap "44"\
      -Access "All" -SysfailReset

      -Name "SOManButt_On3" -SignalType "DO" -Unit "BOARD10" -UnitMap "43"\
      -Access "All" -SysfailReset
#
EIO_COMMAND_TYPE:

      -Name "DataWidth_L" -UnitType "d351_Lean" -DefValue "3" -OrderNr 1\
      -DL_Path "6,20 65 24 01 30 01,C6,1"

      -Name "D351reset_L" -UnitType "d351_Lean" -DefValue "0" -OrderNr 2\
      -DL_Path "4,20 01 24 01,C1,1" -DL_Service 5

      -Name "MasterInputSize_B_L" -UnitType "d352_Lean" -DefValue "1" -OrderNr 1\
      -DL_Path "6,20 67 24 01 30 02,C6,1"

      -Name "MasterOutputSize_B_L" -UnitType "d352_Lean" -DefValue "1"\
      -OrderNr 2 -DL_Path "6,20 67 24 01 30 03,C6,1"

      -Name "StationAddress_B_L" -UnitType "d352_Lean" -DefValue "126"\
      -OrderNr 3 -DL_Path "6,20 67 24 01 30 04,C6,1"

      -Name "D352reset_L" -UnitType "d352_Lean" -DefValue "0" -OrderNr 4\
      -DL_Path "4,20 01 24 01,C1,1" -DL_Service 5

      -Name "StationNo_L" -UnitType "d378_Lean" -DefValue "1" -OrderNr 1\
      -DL_Path "6,20 68 24 01 30 01,C6,1"

      -Name "BaudRate_L" -UnitType "d378_Lean" -DefValue "0" -OrderNr 2\
      -DL_Path "6,20 68 24 01 30 02,C6,1"

      -Name "OccStat_L" -UnitType "d378_Lean" -DefValue "1" -OrderNr 3\
      -DL_Path "6,20 68 24 01 30 03,C6,1"

      -Name "BasicIO_L" -UnitType "d378_Lean" -DefValue "0" -OrderNr 4\
      -DL_Path "6,20 68 24 01 30 04,C1,1"

      -Name "D378reset_L" -UnitType "d378_Lean" -DefValue "0" -OrderNr 5\
      -DL_Path "4,20 01 24 01,C1,1" -DL_Service 5
#
EIO_ACCESS:

      -Name "All" -Rapid  -LocalManual  -LocalAuto  -RemoteManual  -RemoteAuto

--- Backups/120-502354_Topsy/SYSPAR/EIO.cfg ---
EIO:CFG_1.0:5:0::
#
EIO_BUS:

      -Name "Virtual1" -ConnectorID "SIM1"

      -Name "DeviceNet_Lean" -BusType "DNLE" -ConnectorID "PCI1"\
      -ConnectorLabel "DeviceNet Lean"
#
EIO_UNIT_TYPE:

      -Name "Virtual" -VendorName "ABB" -ProductName "Virtual unit"

      -Name "d651_Lean" -BusType "DNLE" -VendorName "ABB Robotics"\
      -ProductName "Combi Unit" -DL_ProductCode 25

      -Name "d652_Lean" -BusType "DNLE" -VendorName "ABB Robotics"\
      -ProductName "24 VDC Unit" -DL_ProductCode 26

      -Name "d653_Lean" -BusType "DNLE" -VendorName "ABB Robotics"\
      -ProductName "Relay Unit" -DL_ProductCode 27

      -Name "AC500_PLC_Lean" -BusType "DNLE" -VendorName "ABB Stotz"\
      -ProductName "AC500 PLC - FPB" -DL_ProductCode 1 -DL_VendorID 760

      -Name "DL_GENERIC" -BusType "DNLE" -DL_ProductCode 3535

      -Name "DL_GENERIC_POLL" -BusType "DNLE" -DL_ProductCode 3535\
      -DL_Pollrate 30

      -Name "d351_Lean" -BusType "DNLE" -VendorName "ABB Robotics"\
      -ProductName "IBS Adapter" -DL_ProductCode 7

      -Name "d352_Lean" -BusType "DNLE" -VendorName "ABB Robotics"\
      -ProductName "PBUS Adapter" -DL_ProductCode 8

      -Name "d378_Lean" -BusType "DNLE" -VendorName "ABB Robotics"\
      -ProductName "CCLink Adapter" -DL_ProductCode 17
#
EIO_UNIT:

      -Name "BOARD10" -UnitType "d652_Lean" -Bus "DeviceNet_Lean" -DL_Address 10
#
EIO_SIGNAL:

      -Name "DI10_1" -SignalType "DI" -Unit "BOARD10" -UnitMap "0"

      -Name "DI10_2" -SignalType "DI" -Unit "BOARD10" -UnitMap "1"

      -Name "DI10_3" -SignalType "DI" -Unit "BOARD10" -UnitMap "2"

      -Name "DI10_4" -SignalType "DI" -Unit "BOARD10" -UnitMap "3"

      -Name "DI10_5" -SignalType "DI" -Unit "BOARD10" -UnitMap "4"

      -Name "DI10_6" -SignalType "DI" -Unit "BOARD10" -UnitMap "5"

      -Name "DI10_7" -SignalType "DI" -Unit "BOARD10" -UnitMap "6"

      -Name "DI10_8" -SignalType "DI" -Unit "BOARD10" -UnitMap "7"

      -Name "DI10_9" -SignalType "DI" -Unit "BOARD10" -UnitMap "8"

      -Name "DI10_10" -SignalType "DI" -Unit "BOARD10" -UnitMap "9"

      -Name "DI10_11" -SignalType "DI" -Unit "BOARD10" -UnitMap "10"

      -Name "DI10_12" -SignalType "DI" -Unit "BOARD10" -UnitMap "11"

      -Name "DI10_13" -SignalType "DI" -Unit "BOARD10" -UnitMap "12"

      -Name "DI10_14" -SignalType "DI" -Unit "BOARD10" -UnitMap "13"

      -Name "DI10_15" -SignalType "DI" -Unit "BOARD10" -UnitMap "14"

      -Name "DI10_16" -SignalType "DI" -Unit "BOARD10" -UnitMap "15"

      -Name "DO10_1" -SignalType "DO" -Unit "BOARD10" -UnitMap "0"

      -Name "DO10_2" -SignalType "DO" -Unit "BOARD10" -UnitMap "1"

      -Name "DO10_3" -SignalType "DO" -Unit "BOARD10" -UnitMap "2"

      -Name "DO10_4" -SignalType "DO" -Unit "BOARD10" -UnitMap "3"

      -Name "DO10_5" -SignalType "DO" -Unit "BOARD10" -UnitMap "4"

      -Name "DO10_6" -SignalType "DO" -Unit "BOARD10" -UnitMap "5"

      -Name "DO10_7" -SignalType "DO" -Unit "BOARD10" -UnitMap "6"

      -Name "DO10_8" -SignalType "DO" -Unit "BOARD10" -UnitMap "7"

      -Name "DO10_9" -SignalType "DO" -Unit "BOARD10" -UnitMap "8"

      -Name "DO10_10" -SignalType "DO" -Unit "BOARD10" -UnitMap "9"

      -Name "DO10_11" -SignalType "DO" -Unit "BOARD10" -UnitMap "10"

      -Name "DO10_12" -SignalType "DO" -Unit "BOARD10" -UnitMap "11"

      -Name "DO10_13" -SignalType "DO" -Unit "BOARD10" -UnitMap "12"

      -Name "DO10_14" -SignalType "DO" -Unit "BOARD10" -UnitMap "13"

      -Name "DO10_15" -SignalType "DO" -Unit "BOARD10" -UnitMap "14"

      -Name "DO10_16" -SignalType "DO" -Unit "BOARD10" -UnitMap "15"

      -Name "SOManButt_On1" -SignalType "DO" -Unit "BOARD10" -UnitMap "41"\
      -Access "All" -SysfailReset

      -Name "SOManButt_On2" -SignalType "DO" -Unit "BOARD10" -UnitMap "42"\
      -Access "All" -SysfailReset

      -Name "SOManButt_On3" -SignalType "DO" -Unit "BOARD10" -UnitMap "43"\
      -Access "All" -SysfailReset

      -Name "SOManButt_On4" -SignalType "DO" -Unit "BOARD10" -UnitMap "44"\
      -Access "All" -SysfailReset
#
EIO_COMMAND_TYPE:

      -Name "DataWidth_L" -UnitType "d351_Lean" -DefValue "3" -OrderNr 1\
      -DL_Path "6,20 65 24 01 30 01,C6,1"

      -Name "D351reset_L" -UnitType "d351_Lean" -DefValue "0" -OrderNr 2\
      -DL_Path "4,20 01 24 01,C1,1" -DL_Service 5

      -Name "MasterInputSize_B_L" -UnitType "d352_Lean" -DefValue "1" -OrderNr 1\
      -DL_Path "6,20 67 24 01 30 02,C6,1"

      -Name "MasterOutputSize_B_L" -UnitType "d352_Lean" -DefValue "1"\
      -OrderNr 2 -DL_Path "6,20 67 24 01 30 03,C6,1"

      -Name "StationAddress_B_L" -UnitType "d352_Lean" -DefValue "126"\
      -OrderNr 3 -DL_Path "6,20 67 24 01 30 04,C6,1"

      -Name "D352reset_L" -UnitType "d352_Lean" -DefValue "0" -OrderNr 4\
      -DL_Path "4,20 01 24 01,C1,1" -DL_Service 5

      -Name "StationNo_L" -UnitType "d378_Lean" -DefValue "1" -OrderNr 1\
      -DL_Path "6,20 68 24 01 30 01,C6,1"

      -Name "BaudRate_L" -UnitType "d378_Lean" -DefValue "0" -OrderNr 2\
      -DL_Path "6,20 68 24 01 30 02,C6,1"

      -Name "OccStat_L" -UnitType "d378_Lean" -DefValue "1" -OrderNr 3\
      -DL_Path "6,20 68 24 01 30 03,C6,1"

      -Name "BasicIO_L" -UnitType "d378_Lean" -DefValue "0" -OrderNr 4\
      -DL_Path "6,20 68 24 01 30 04,C1,1"

      -Name "D378reset_L" -UnitType "d378_Lean" -DefValue "0" -OrderNr 5\
      -DL_Path "4,20 01 24 01,C1,1" -DL_Service 5
#
EIO_ACCESS:

      -Name "All" -Rapid  -LocalManual  -LocalAuto  -RemoteManual  -RemoteAuto
